   LIN {X 9.682, Y 0.522, Z 73.100}
   LaserStart_Ext()
   LIN {X -1.874, Y 0.522, Z 73.100}
   LaserEnd_Ext()
   LIN {X -2.025, Y -0.478, Z 73.100}
   LaserStart_Ext()
   LIN {X 9.715, Y -0.478, Z 73.100}
   LaserEnd_Ext()
   LIN {X 9.743, Y -1.478, Z 73.100}
   LaserStart_Ext()
   LIN {X -2.174, Y -1.478, Z 73.100}
   LaserEnd_Ext()
   LIN {X -2.322, Y -2.478, Z 73.100}
   LaserStart_Ext()
   LIN {X 9.770, Y -2.478, Z 73.100}
   LaserEnd_Ext()
   LIN {X 9.797, Y -3.478, Z 73.100}
   LaserStart_Ext()
   LIN {X -2.486, Y -3.478, Z 73.100}
   LaserEnd_Ext()
   LIN {X -2.718, Y -4.478, Z 73.100}
   LaserStart_Ext()
   LIN {X 9.824, Y -4.478, Z 73.100}
   LaserEnd_Ext()
   LIN {X 9.851, Y -5.478, Z 73.100}
   LaserStart_Ext()
   LIN {X -2.954, Y -5.478, Z 73.100}
   LaserEnd_Ext()
   LIN {X -3.189, Y -6.478, Z 73.100}
   LaserStart_Ext()
   LIN {X 9.859, Y -6.478, Z 73.100}
   LaserEnd_Ext()
   LIN {X 9.835, Y -7.478, Z 73.100}
   LaserStart_Ext()
   LIN {X -3.425, Y -7.478, Z 73.100}
   LaserEnd_Ext()
   LIN {X -3.704, Y -8.478, Z 73.100}
   LaserStart_Ext()
   LIN {X 9.811, Y -8.478, Z 73.100}
   LaserEnd_Ext()
   LIN {X 9.787, Y -9.478, Z 73.100}
   LaserStart_Ext()
   LIN {X -4.012, Y -9.478, Z 73.100}
   LaserEnd_Ext()
   LIN {X -4.320, Y -10.478, Z 73.100}
   LaserStart_Ext()
   LIN {X 9.763, Y -10.478, Z 73.100}
   LaserEnd_Ext()
   LIN {X 9.717, Y -11.478, Z 73.100}
   LaserStart_Ext()
   LIN {X -4.621, Y -11.478, Z 73.100}
   LaserEnd_Ext()
   LIN {X -4.914, Y -12.478, Z 73.100}
   LaserStart_Ext()
   LIN {X 9.656, Y -12.478, Z 73.100}
   LaserEnd_Ext()
   LIN {X 9.594, Y -13.478, Z 73.100}
   LaserStart_Ext()
   LIN {X -5.269, Y -13.478, Z 73.100}
   LaserEnd_Ext()
   LIN {X -5.652, Y -14.478, Z 73.100}
   LaserStart_Ext()
   LIN {X -1.831, Y -14.478, Z 73.100}
   LaserEnd_Ext()
   LIN {X 3.606, Y -14.478, Z 73.100}
   LaserStart_Ext()
   LIN {X 9.526, Y -14.478, Z 73.100}
   LaserEnd_Ext()
   LIN {X 9.435, Y -15.478, Z 73.100}
   LaserStart_Ext()
   LIN {X 5.099, Y -15.478, Z 73.100}
   LaserEnd_Ext()
   LIN {X -3.147, Y -15.478, Z 73.100}
   LaserStart_Ext()
   LIN {X -6.034, Y -15.478, Z 73.100}
   LaserEnd_Ext()
   LIN {X -6.409, Y -16.478, Z 73.100}
   LaserStart_Ext()
   LIN {X -4.119, Y -16.478, Z 73.100}
   LaserEnd_Ext()
   LIN {X 5.774, Y -16.478, Z 73.100}
   LaserStart_Ext()
   LIN {X 9.340, Y -16.478, Z 73.100}
   LaserEnd_Ext()
   LIN {X 9.248, Y -17.478, Z 73.100}
   LaserStart_Ext()
   LIN {X 6.448, Y -17.478, Z 73.100}
   LaserEnd_Ext()
   LIN {X -4.449, Y -17.478, Z 73.100}
   LaserStart_Ext()
   LIN {X -6.647, Y -17.478, Z 73.100}
   LaserEnd_Ext()
   LIN {X -6.866, Y -18.478, Z 73.100}
   LaserStart_Ext()
   LIN {X -4.737, Y -18.478, Z 73.100}
   LaserEnd_Ext()
   LIN {X 6.690, Y -18.478, Z 73.100}
   LaserStart_Ext()
   LIN {X 9.132, Y -18.478, Z 73.100}
   LaserEnd_Ext()
   LIN {X 9.008, Y -19.478, Z 73.100}
   LaserStart_Ext()
   LIN {X 6.800, Y -19.478, Z 73.100}
   LaserEnd_Ext()
   LIN {X -5.030, Y -19.478, Z 73.100}
   LaserStart_Ext()
   LIN {X -7.084, Y -19.478, Z 73.100}
   LaserEnd_Ext()
   LIN {X -6.914, Y -20.478, Z 73.100}
   LaserStart_Ext()
   LIN {X -4.983, Y -20.478, Z 73.100}
   LaserEnd_Ext()
   LIN {X 6.856, Y -20.478, Z 73.100}
   LaserStart_Ext()
   LIN {X 8.885, Y -20.478, Z 73.100}
   LaserEnd_Ext()
   LIN {X 8.615, Y -21.478, Z 73.100}
   LaserStart_Ext()
   LIN {X 6.497, Y -21.478, Z 73.100}
   LaserEnd_Ext()
   LIN {X -4.753, Y -21.478, Z 73.100}
   LaserStart_Ext()
   LIN {X -6.741, Y -21.478, Z 73.100}
   LaserEnd_Ext()
   LIN {X -6.568, Y -22.478, Z 73.100}
   LaserStart_Ext()
   LIN {X -4.439, Y -22.478, Z 73.100}
   LaserEnd_Ext()
   LIN {X 6.127, Y -22.478, Z 73.100}
   LaserStart_Ext()
   LIN {X 8.304, Y -22.478, Z 73.100}
   LaserEnd_Ext()
   LIN {X 7.905, Y -23.478, Z 73.100}
   LaserStart_Ext()
   LIN {X 5.494, Y -23.478, Z 73.100}
   LaserEnd_Ext()
   LIN {X -3.676, Y -23.478, Z 73.100}
   LaserStart_Ext()
   LIN {X -6.049, Y -23.478, Z 73.100}
   LaserEnd_Ext()
   LIN {X -5.411, Y -24.478, Z 73.100}
   LaserStart_Ext()
   LIN {X -2.745, Y -24.478, Z 73.100}
   LaserEnd_Ext()
   LIN {X 4.468, Y -24.478, Z 73.100}
   LaserStart_Ext()
   LIN {X 7.178, Y -24.478, Z 73.100}
   LaserEnd_Ext()
   LIN {X 6.380, Y -25.478, Z 73.100}
   LaserStart_Ext()
   LIN {X 2.288, Y -25.478, Z 73.100}
   LaserEnd_Ext()
   LIN {X -0.890, Y -25.478, Z 73.100}
   LaserStart_Ext()
   LIN {X -4.635, Y -25.478, Z 73.100}
   LaserEnd_Ext()
   LIN {X -3.321, Y -26.478, Z 73.100}
   LaserStart_Ext()
   LIN {X 4.795, Y -26.478, Z 73.100}
   LaserEnd_Ext()
   LIN {X 2.332, Y -27.478, Z 73.100}
   LaserStart_Ext()
   LIN {X -0.220, Y -27.478, Z 73.100}
   LaserEnd_Ext()
   LIN {X 5.714, Y -18.002, Z 73.950}
   LaserStart_Ext()
   LIN {X 5.782, Y -18.621, Z 73.950} C_DIS
   LIN {X 5.961, Y -20.198, Z 73.950} C_DIS
   LIN {X 5.569, Y -21.275, Z 73.950} C_DIS
   LIN {X 5.134, Y -22.450, Z 73.950} C_DIS
   LIN {X 3.676, Y -23.879, Z 73.950} C_DIS
   LIN {X 1.580, Y -24.646, Z 73.950} C_DIS
   LIN {X 0.264, Y -24.545, Z 73.950} C_DIS
   LIN {X -0.466, Y -24.486, Z 73.950} C_DIS
   LIN {X -1.367, Y -23.994, Z 73.950} C_DIS
   LIN {X -2.280, Y -23.497, Z 73.950} C_DIS
   LIN {X -2.814, Y -22.805, Z 73.950} C_DIS
   LIN {X -3.548, Y -21.845, Z 73.950} C_DIS
   LIN {X -3.815, Y -20.687, Z 73.950} C_DIS
   LIN {X -4.019, Y -19.812, Z 73.950} C_DIS
   LIN {X -3.359, Y -17.520, Z 73.950} C_DIS
   LIN {X -3.209, Y -16.978, Z 73.950} C_DIS
   LIN {X -2.651, Y -16.408, Z 73.950} C_DIS
   LIN {X -1.744, Y -15.500, Z 73.950} C_DIS
   LIN {X -0.780, Y -15.138, Z 73.950} C_DIS
   LIN {X 0.268, Y -14.732, Z 73.950} C_DIS
   LIN {X 1.745, Y -14.827, Z 73.950} C_DIS
   LIN {X 2.426, Y -14.872, Z 73.950} C_DIS
   LIN {X 2.906, Y -15.138, Z 73.950} C_DIS
   LIN {X 4.288, Y -15.897, Z 73.950} C_DIS
   LIN {X 5.367, Y -17.486, Z 73.950} C_DIS
   LIN {X 5.714, Y -18.002, Z 73.950}
   LaserEnd_Ext()
   LIN {X -4.465, Y 29.728, Z 73.950}
   LaserStart_Ext()
   LIN {X -4.338, Y 29.252, Z 73.950} C_DIS
   LIN {X -3.932, Y 27.798, Z 73.950} C_DIS
   LIN {X -3.385, Y 25.231, Z 73.950} C_DIS
   LIN {X -3.010, Y 22.795, Z 73.950} C_DIS
   LIN {X -2.537, Y 19.684, Z 73.950} C_DIS
   LIN {X -2.269, Y 17.163, Z 73.950} C_DIS
   LIN {X -2.334, Y 9.229, Z 73.950} C_DIS
   LIN {X -2.281, Y 5.034, Z 73.950} C_DIS
   LIN {X -2.382, Y 3.614, Z 73.950} C_DIS
   LIN {X -3.332, Y -2.684, Z 73.950} C_DIS
   LIN {X -3.464, Y -3.444, Z 73.950} C_DIS
   LIN {X -3.710, Y -4.444, Z 73.950} C_DIS
   LIN {X -4.539, Y -7.966, Z 73.950} C_DIS
   LIN {X -5.833, Y -12.173, Z 73.950} C_DIS
   LIN {X -5.930, Y -12.505, Z 73.950} C_DIS
   LIN {X -6.001, Y -12.710, Z 73.950} C_DIS
   LIN {X -6.189, Y -13.202, Z 73.950} C_DIS
   LIN {X -7.363, Y -16.331, Z 73.950} C_DIS
   LIN {X -7.756, Y -18.196, Z 73.950} C_DIS
   LIN {X -8.026, Y -19.431, Z 73.950} C_DIS
   LIN {X -7.590, Y -21.953, Z 73.950} C_DIS
   LIN {X -7.388, Y -23.087, Z 73.950} C_DIS
   LIN {X -7.016, Y -23.696, Z 73.950} C_DIS
   LIN {X -5.673, Y -25.799, Z 73.950} C_DIS
   LIN {X -4.232, Y -26.896, Z 73.950} C_DIS
   LIN {X -3.323, Y -27.631, Z 73.950} C_DIS
   LIN {X -2.826, Y -27.851, Z 73.950} C_DIS
   LIN {X 0.153, Y -28.583, Z 73.950} C_DIS
   LIN {X 0.920, Y -28.695, Z 73.950} C_DIS
   LIN {X 2.776, Y -28.357, Z 73.950} C_DIS
   LIN {X 4.021, Y -28.148, Z 73.950} C_DIS
   LIN {X 4.653, Y -27.762, Z 73.950} C_DIS
   LIN {X 7.309, Y -26.062, Z 73.950} C_DIS
   LIN {X 8.675, Y -24.178, Z 73.950} C_DIS
   LIN {X 9.048, Y -23.657, Z 73.950} C_DIS
   LIN {X 9.328, Y -22.743, Z 73.950} C_DIS
   LIN {X 9.923, Y -20.827, Z 73.950} C_DIS
   LIN {X 10.086, Y -19.502, Z 73.950} C_DIS
   LIN {X 10.310, Y -17.587, Z 73.950} C_DIS
   LIN {X 10.557, Y -14.882, Z 73.950} C_DIS
   LIN {X 10.580, Y -14.638, Z 73.950} C_DIS
   LIN {X 10.593, Y -14.454, Z 73.950} C_DIS
   LIN {X 10.811, Y -10.839, Z 73.950} C_DIS
   LIN {X 10.890, Y -7.567, Z 73.950} C_DIS
   LIN {X 10.916, Y -6.053, Z 73.950} C_DIS
   LIN {X 10.830, Y -3.422, Z 73.950} C_DIS
   LIN {X 10.724, Y 0.460, Z 73.950} C_DIS
   LIN {X 10.682, Y 1.154, Z 73.950} C_DIS
   LIN {X 10.578, Y 2.845, Z 73.950} C_DIS
   LIN {X 9.965, Y 8.271, Z 73.950} C_DIS
   LIN {X 9.810, Y 9.484, Z 73.950} C_DIS
   LIN {X 9.543, Y 10.719, Z 73.950} C_DIS
   LIN {X 7.636, Y 20.594, Z 73.950} C_DIS
   LIN {X 6.675, Y 24.247, Z 73.950} C_DIS
   LIN {X 5.389, Y 28.268, Z 73.950} C_DIS
   LIN {X 4.625, Y 30.707, Z 73.950} C_DIS
   LIN {X 3.858, Y 32.710, Z 73.950} C_DIS
   LIN {X 3.063, Y 34.855, Z 73.950} C_DIS
   LIN {X 2.554, Y 36.078, Z 73.950} C_DIS
   LIN {X 1.908, Y 37.651, Z 73.950} C_DIS
   LIN {X 0.727, Y 40.299, Z 73.950} C_DIS
   LIN {X 0.658, Y 40.450, Z 73.950} C_DIS
   LIN {X -0.114, Y 42.085, Z 73.950} C_DIS
   LIN {X -0.641, Y 43.162, Z 73.950} C_DIS
   LIN {X -0.767, Y 43.418, Z 73.950} C_DIS
   LIN {X -1.000, Y 43.725, Z 73.950} C_DIS
   LIN {X -1.653, Y 44.592, Z 73.950} C_DIS
   LIN {X -2.406, Y 45.027, Z 73.950} C_DIS
   LIN {X -3.161, Y 45.460, Z 73.950} C_DIS
   LIN {X -4.407, Y 45.564, Z 73.950} C_DIS
   LIN {X -4.900, Y 45.607, Z 73.950} C_DIS
   LIN {X -6.040, Y 44.979, Z 73.950} C_DIS
   LIN {X -7.379, Y 44.245, Z 73.950} C_DIS
   LIN {X -7.707, Y 43.622, Z 73.950} C_DIS
   LIN {X -8.206, Y 42.649, Z 73.950} C_DIS
   LIN {X -8.267, Y 41.850, Z 73.950} C_DIS
   LIN {X -8.311, Y 41.308, Z 73.950} C_DIS
   LIN {X -8.222, Y 40.974, Z 73.950} C_DIS
   LIN {X -7.991, Y 40.080, Z 73.950} C_DIS
   LIN {X -7.513, Y 38.929, Z 73.950} C_DIS
   LIN {X -6.918, Y 37.439, Z 73.950} C_DIS
   LIN {X -6.145, Y 35.340, Z 73.950} C_DIS
   LIN {X -6.099, Y 35.214, Z 73.950} C_DIS
   LIN {X -6.060, Y 35.097, Z 73.950} C_DIS
   LIN {X -5.193, Y 32.448, Z 73.950} C_DIS
   LIN {X -4.849, Y 31.163, Z 73.950} C_DIS
   LIN {X -4.593, Y 30.206, Z 73.950} C_DIS
   LIN {X -4.465, Y 29.728, Z 73.950}
   LaserEnd_Ext()
   LIN {X -7.280, Y 41.321, Z 73.950}
   LaserStart_Ext()
   LIN {X -7.280, Y 41.655, Z 73.950}
   LaserEnd_Ext()
   LIN {X -6.280, Y 43.707, Z 73.950}
   LaserStart_Ext()
   LIN {X -6.280, Y 38.538, Z 73.950}
   LaserEnd_Ext()
   LIN {X -6.280, Y -16.290, Z 73.950}
   LaserStart_Ext()
   LIN {X -6.280, Y -22.983, Z 73.950}
   LaserEnd_Ext()
   LIN {X -5.280, Y -24.557, Z 73.950}
   LaserStart_Ext()
   LIN {X -5.280, Y -13.624, Z 73.950}
   LaserEnd_Ext()
   LIN {X -5.280, Y 35.884, Z 73.950}
   LaserStart_Ext()
   LIN {X -5.280, Y 44.256, Z 73.950}
   LaserEnd_Ext()
   LIN {X -4.280, Y 44.550, Z 73.950}
   LaserStart_Ext()
   LIN {X -4.280, Y 32.874, Z 73.950}
   LaserEnd_Ext()
   LIN {X -4.280, Y -10.525, Z 73.950}
   LaserStart_Ext()
   LIN {X -4.280, Y -17.099, Z 73.950}
   LaserEnd_Ext()
   LIN {X -4.280, Y -22.535, Z 73.950}
   LaserStart_Ext()
   LIN {X -4.280, Y -25.603, Z 73.950}
   LaserEnd_Ext()
   LIN {X -3.280, Y -26.380, Z 73.950}
   LaserStart_Ext()
   LIN {X -3.280, Y -23.838, Z 73.950}
   LaserEnd_Ext()
   LIN {X -3.280, Y -15.623, Z 73.950}
   LaserStart_Ext()
   LIN {X -3.280, Y -6.982, Z 73.950}
   LaserEnd_Ext()
   LIN {X -3.280, Y 29.182, Z 73.950}
   LaserStart_Ext()
   LIN {X -3.280, Y 44.375, Z 73.950}
   LaserEnd_Ext()
   LIN {X -2.280, Y 43.762, Z 73.950}
   LaserStart_Ext()
   LIN {X -2.280, Y 24.625, Z 73.950}
   LaserEnd_Ext()
   LIN {X -2.280, Y -2.415, Z 73.950}
   LaserStart_Ext()
   LIN {X -2.280, Y -14.656, Z 73.950}
   LaserEnd_Ext()
   LIN {X -2.280, Y -24.636, Z 73.950}
   LaserStart_Ext()
   LIN {X -2.280, Y -26.955, Z 73.950}
   LaserEnd_Ext()
   LIN {X -1.280, Y -27.201, Z 73.950}
   LaserStart_Ext()
   LIN {X -1.280, Y -25.181, Z 73.950}
   LaserEnd_Ext()
   LIN {X -1.280, Y -14.257, Z 73.950}
   LaserStart_Ext()
   LIN {X -1.280, Y 15.884, Z 73.950}
   LaserEnd_Ext()
   LIN {X -1.280, Y 17.314, Z 73.950}
   LaserStart_Ext()
   LIN {X -1.280, Y 42.193, Z 73.950}
   LaserEnd_Ext()
   LIN {X -0.280, Y 40.094, Z 73.950}
   LaserStart_Ext()
   LIN {X -0.280, Y -13.872, Z 73.950}
   LaserEnd_Ext()
   LIN {X -0.280, Y -25.504, Z 73.950}
   LaserStart_Ext()
   LIN {X -0.280, Y -27.447, Z 73.950}
   LaserEnd_Ext()
   LIN {X 0.720, Y -27.655, Z 73.950}
   LaserStart_Ext()
   LIN {X 0.720, Y -25.583, Z 73.950}
   LaserEnd_Ext()
   LIN {X 0.720, Y -13.759, Z 73.950}
   LaserStart_Ext()
   LIN {X 0.720, Y 37.859, Z 73.950}
   LaserEnd_Ext()
   LIN {X 1.720, Y 35.480, Z 73.950}
   LaserStart_Ext()
   LIN {X 1.720, Y -13.823, Z 73.950}
   LaserEnd_Ext()
   LIN {X 1.720, Y -25.635, Z 73.950}
   LaserStart_Ext()
   LIN {X 1.720, Y -27.533, Z 73.950}
   LaserEnd_Ext()
   LIN {X 2.720, Y -27.352, Z 73.950}
   LaserStart_Ext()
   LIN {X 2.720, Y -25.298, Z 73.950}
   LaserEnd_Ext()
   LIN {X 2.720, Y -13.917, Z 73.950}
   LaserStart_Ext()
   LIN {X 2.720, Y 32.902, Z 73.950}
   LaserEnd_Ext()
   LIN {X 3.720, Y 30.251, Z 73.950}
   LaserStart_Ext()
   LIN {X 3.720, Y -14.444, Z 73.950}
   LaserEnd_Ext()
   LIN {X 3.720, Y -24.939, Z 73.950}
   LaserStart_Ext()
   LIN {X 3.720, Y -27.160, Z 73.950}
   LaserEnd_Ext()
   LIN {X 4.720, Y -26.532, Z 73.950}
   LaserStart_Ext()
   LIN {X 4.720, Y -24.256, Z 73.950}
   LaserEnd_Ext()
   LIN {X 4.720, Y -14.993, Z 73.950}
   LaserStart_Ext()
   LIN {X 4.720, Y 27.077, Z 73.950}
   LaserEnd_Ext()
   LIN {X 5.720, Y 23.946, Z 73.950}
   LaserStart_Ext()
   LIN {X 5.720, Y -16.226, Z 73.950}
   LaserEnd_Ext()
   LIN {X 5.720, Y -23.276, Z 73.950}
   LaserStart_Ext()
   LIN {X 5.720, Y -25.892, Z 73.950}
   LaserEnd_Ext()
   LIN {X 6.720, Y -25.171, Z 73.950}
   LaserStart_Ext()
   LIN {X 6.720, Y -21.036, Z 73.950}
   LaserEnd_Ext()
   LIN {X 6.720, Y -18.000, Z 73.950}
   LaserStart_Ext()
   LIN {X 6.720, Y 20.065, Z 73.950}
   LaserEnd_Ext()
   LIN {X 7.720, Y 14.884, Z 73.950}
   LaserStart_Ext()
   LIN {X 7.720, Y -23.791, Z 73.950}
   LaserEnd_Ext()
   LIN {X 8.720, Y -21.328, Z 73.950}
   LaserStart_Ext()
   LIN {X 8.720, Y 9.793, Z 73.950}
   LaserEnd_Ext()
   LIN {X 9.720, Y 0.498, Z 73.950}
   LaserStart_Ext()
   LIN {X 9.720, Y -12.314, Z 73.950}
   LaserEnd_Ext()
   LIN {X -3.144, Y -16.947, Z 74.800}
   LaserStart_Ext()
   LIN {X -1.831, Y -15.605, Z 74.800} C_DIS
   LIN {X -1.699, Y -15.468, Z 74.800} C_DIS
   LIN {X -1.436, Y -15.366, Z 74.800} C_DIS
   LIN {X 0.340, Y -14.679, Z 74.800} C_DIS
   LIN {X 1.732, Y -14.768, Z 74.800} C_DIS
   LIN {X 2.494, Y -14.814, Z 74.800} C_DIS
   LIN {X 3.293, Y -15.250, Z 74.800} C_DIS
   LIN {X 4.358, Y -15.835, Z 74.800} C_DIS
   LIN {X 5.158, Y -17.013, Z 74.800} C_DIS
   LIN {X 5.790, Y -17.936, Z 74.800} C_DIS
   LIN {X 5.889, Y -18.780, Z 74.800} C_DIS
   LIN {X 6.042, Y -20.132, Z 74.800} C_DIS
   LIN {X 5.244, Y -22.323, Z 74.800} C_DIS
   LIN {X 5.147, Y -22.457, Z 74.800} C_DIS
   LIN {X 3.744, Y -23.839, Z 74.800} C_DIS
   LIN {X 2.518, Y -24.284, Z 74.800} C_DIS
   LIN {X 1.668, Y -24.590, Z 74.800} C_DIS
   LIN {X 0.375, Y -24.491, Z 74.800} C_DIS
   LIN {X -0.375, Y -24.435, Z 74.800} C_DIS
   LIN {X -0.865, Y -24.171, Z 74.800} C_DIS
   LIN {X -2.192, Y -23.450, Z 74.800} C_DIS
   LIN {X -3.292, Y -22.022, Z 74.800} C_DIS
   LIN {X -3.464, Y -21.801, Z 74.800} C_DIS
   LIN {X -3.524, Y -21.549, Z 74.800} C_DIS
   LIN {X -3.940, Y -19.770, Z 74.800} C_DIS
   LIN {X -3.577, Y -18.513, Z 74.800} C_DIS
   LIN {X -3.144, Y -16.947, Z 74.800}
   LaserEnd_Ext()
   LIN {X -7.948, Y -19.398, Z 74.800}
   LaserStart_Ext()
   LIN {X -7.855, Y -19.936, Z 74.800} C_DIS
   LIN {X -7.301, Y -23.052, Z 74.800} C_DIS
   LIN {X -6.276, Y -24.727, Z 74.800} C_DIS
   LIN {X -5.697, Y -25.635, Z 74.800} C_DIS
   LIN {X -5.075, Y -26.108, Z 74.800} C_DIS
   LIN {X -3.295, Y -27.549, Z 74.800} C_DIS
   LIN {X -2.320, Y -27.979, Z 74.800} C_DIS
   LIN {X -0.748, Y -28.365, Z 74.800} C_DIS
   LIN {X 1.120, Y -28.639, Z 74.800} C_DIS
   LIN {X 3.648, Y -28.178, Z 74.800} C_DIS
   LIN {X 4.125, Y -28.085, Z 74.800} C_DIS
   LIN {X 5.363, Y -27.299, Z 74.800} C_DIS
   LIN {X 7.404, Y -25.993, Z 74.800} C_DIS
   LIN {X 8.053, Y -25.097, Z 74.800} C_DIS
   LIN {X 9.137, Y -23.583, Z 74.800} C_DIS
   LIN {X 9.950, Y -20.927, Z 74.800} C_DIS
   LIN {X 10.005, Y -20.752, Z 74.800} C_DIS
   LIN {X 10.020, Y -20.630, Z 74.800} C_DIS
   LIN {X 10.384, Y -17.510, Z 74.800} C_DIS
   LIN {X 10.556, Y -15.630, Z 74.800} C_DIS
   LIN {X 10.648, Y -14.561, Z 74.800} C_DIS
   LIN {X 10.747, Y -12.799, Z 74.800} C_DIS
   LIN {X 10.870, Y -10.762, Z 74.800} C_DIS
   LIN {X 10.909, Y -9.133, Z 74.800} C_DIS
   LIN {X 10.963, Y -5.975, Z 74.800} C_DIS
   LIN {X 10.784, Y -0.487, Z 74.800} C_DIS
   LIN {X 10.757, Y 0.537, Z 74.800} C_DIS
   LIN {X 10.745, Y 0.721, Z 74.800} C_DIS
   LIN {X 10.632, Y 2.561, Z 74.800} C_DIS
   LIN {X 10.112, Y 7.163, Z 74.800} C_DIS
   LIN {X 9.771, Y 9.841, Z 74.800} C_DIS
   LIN {X 9.180, Y 12.567, Z 74.800} C_DIS
   LIN {X 7.599, Y 20.760, Z 74.800} C_DIS
   LIN {X 6.801, Y 23.790, Z 74.800} C_DIS
   LIN {X 5.734, Y 27.126, Z 74.800} C_DIS
   LIN {X 4.623, Y 30.674, Z 74.800} C_DIS
   LIN {X 3.507, Y 33.588, Z 74.800} C_DIS
   LIN {X 3.024, Y 34.892, Z 74.800} C_DIS
   LIN {X 2.104, Y 37.104, Z 74.800} C_DIS
   LIN {X 1.928, Y 37.532, Z 74.800} C_DIS
   LIN {X 1.581, Y 38.309, Z 74.800} C_DIS
   LIN {X 0.644, Y 40.402, Z 74.800} C_DIS
   LIN {X -0.104, Y 41.979, Z 74.800} C_DIS
   LIN {X -0.179, Y 42.136, Z 74.800} C_DIS
   LIN {X -0.266, Y 42.313, Z 74.800} C_DIS
   LIN {X -0.835, Y 43.468, Z 74.800} C_DIS
   LIN {X -1.397, Y 44.210, Z 74.800} C_DIS
   LIN {X -1.724, Y 44.640, Z 74.800} C_DIS
   LIN {X -2.393, Y 45.022, Z 74.800} C_DIS
   LIN {X -3.234, Y 45.504, Z 74.800} C_DIS
   LIN {X -3.928, Y 45.563, Z 74.800} C_DIS
   LIN {X -4.973, Y 45.647, Z 74.800} C_DIS
   LIN {X -6.690, Y 44.715, Z 74.800} C_DIS
   LIN {X -7.418, Y 44.316, Z 74.800} C_DIS
   LIN {X -7.716, Y 43.749, Z 74.800} C_DIS
   LIN {X -8.254, Y 42.753, Z 74.800} C_DIS
   LIN {X -8.323, Y 41.939, Z 74.800} C_DIS
   LIN {X -8.372, Y 41.322, Z 74.800} C_DIS
   LIN {X -8.169, Y 40.552, Z 74.800} C_DIS
   LIN {X -8.051, Y 40.112, Z 74.800} C_DIS
   LIN {X -7.913, Y 39.782, Z 74.800} C_DIS
   LIN {X -7.568, Y 38.959, Z 74.800} C_DIS
   LIN {X -7.062, Y 37.699, Z 74.800} C_DIS
   LIN {X -6.972, Y 37.474, Z 74.800} C_DIS
   LIN {X -6.886, Y 37.245, Z 74.800} C_DIS
   LIN {X -6.148, Y 35.252, Z 74.800} C_DIS
   LIN {X -5.378, Y 32.924, Z 74.800} C_DIS
   LIN {X -5.235, Y 32.487, Z 74.800} C_DIS
   LIN {X -5.179, Y 32.276, Z 74.800} C_DIS
   LIN {X -4.827, Y 30.959, Z 74.800} C_DIS
   LIN {X -4.651, Y 30.303, Z 74.800} C_DIS
   LIN {X -4.475, Y 29.647, Z 74.800} C_DIS
   LIN {X -3.917, Y 27.648, Z 74.800} C_DIS
   LIN {X -3.438, Y 25.397, Z 74.800} C_DIS
   LIN {X -2.758, Y 20.982, Z 74.800} C_DIS
   LIN {X -2.456, Y 18.992, Z 74.800} C_DIS
   LIN {X -2.284, Y 17.379, Z 74.800} C_DIS
   LIN {X -2.326, Y 12.303, Z 74.800} C_DIS
   LIN {X -2.239, Y 5.526, Z 74.800} C_DIS
   LIN {X -2.403, Y 3.231, Z 74.800} C_DIS
   LIN {X -3.187, Y -1.972, Z 74.800} C_DIS
   LIN {X -3.508, Y -3.811, Z 74.800} C_DIS
   LIN {X -4.102, Y -6.230, Z 74.800} C_DIS
   LIN {X -4.597, Y -8.330, Z 74.800} C_DIS
   LIN {X -5.563, Y -11.471, Z 74.800} C_DIS
   LIN {X -5.912, Y -12.599, Z 74.800} C_DIS
   LIN {X -6.221, Y -13.443, Z 74.800} C_DIS
   LIN {X -7.292, Y -16.296, Z 74.800} C_DIS
   LIN {X -7.890, Y -19.135, Z 74.800} C_DIS
   LIN {X -7.948, Y -19.398, Z 74.800}
   LaserEnd_Ext()
   LIN {X -0.648, Y -27.360, Z 74.800}
   LaserStart_Ext()
   LIN {X 2.557, Y -27.360, Z 74.800}
   LaserEnd_Ext()
   LIN {X 4.975, Y -26.360, Z 74.800}
   LaserStart_Ext()
   LIN {X -3.174, Y -26.360, Z 74.800}
   LaserEnd_Ext()
   LIN {X -4.410, Y -25.360, Z 74.800}
   LaserStart_Ext()
   LIN {X -0.756, Y -25.360, Z 74.800}
   LaserEnd_Ext()
   LIN {X 2.482, Y -25.360, Z 74.800}
   LaserStart_Ext()
   LIN {X 6.537, Y -25.360, Z 74.800}
   LaserEnd_Ext()
   LIN {X 7.351, Y -24.360, Z 74.800}
   LaserStart_Ext()
   LIN {X 4.640, Y -24.360, Z 74.800}
   LaserEnd_Ext()
   LIN {X -2.612, Y -24.360, Z 74.800}
   LaserStart_Ext()
   LIN {X -5.325, Y -24.360, Z 74.800}
   LaserEnd_Ext()
   LIN {X -5.940, Y -23.360, Z 74.800}
   LaserStart_Ext()
   LIN {X -3.524, Y -23.360, Z 74.800}
   LaserEnd_Ext()
   LIN {X 5.655, Y -23.360, Z 74.800}
   LaserStart_Ext()
   LIN {X 8.067, Y -23.360, Z 74.800}
   LaserEnd_Ext()
   LIN {X 8.466, Y -22.360, Z 74.800}
   LaserStart_Ext()
   LIN {X 6.295, Y -22.360, Z 74.800}
   LaserEnd_Ext()
   LIN {X -4.292, Y -22.360, Z 74.800}
   LaserStart_Ext()
   LIN {X -6.408, Y -22.360, Z 74.800}
   LaserEnd_Ext()
   LIN {X -6.586, Y -21.360, Z 74.800}
   LaserStart_Ext()
   LIN {X -4.595, Y -21.360, Z 74.800}
   LaserEnd_Ext()
   LIN {X 6.659, Y -21.360, Z 74.800}
   LaserStart_Ext()
   LIN {X 8.772, Y -21.360, Z 74.800}
   LaserEnd_Ext()
   LIN {X 9.045, Y -20.360, Z 74.800}
   LaserStart_Ext()
   LIN {X 7.014, Y -20.360, Z 74.800}
   LaserEnd_Ext()
   LIN {X -4.829, Y -20.360, Z 74.800}
   LaserStart_Ext()
   LIN {X -6.764, Y -20.360, Z 74.800}
   LaserEnd_Ext()
   LIN {X -6.916, Y -19.360, Z 74.800}
   LaserStart_Ext()
   LIN {X -4.862, Y -19.360, Z 74.800}
   LaserEnd_Ext()
   LIN {X 6.961, Y -19.360, Z 74.800}
   LaserStart_Ext()
   LIN {X 9.161, Y -19.360, Z 74.800}
   LaserEnd_Ext()
   LIN {X 9.278, Y -18.360, Z 74.800}
   LaserStart_Ext()
   LIN {X 6.846, Y -18.360, Z 74.800}
   LaserEnd_Ext()
   LIN {X -4.574, Y -18.360, Z 74.800}
   LaserStart_Ext()
   LIN {X -6.705, Y -18.360, Z 74.800}
   LaserEnd_Ext()
   LIN {X -6.494, Y -17.360, Z 74.800}
   LaserStart_Ext()
   LIN {X -4.296, Y -17.360, Z 74.800}
   LaserEnd_Ext()
   LIN {X 6.608, Y -17.360, Z 74.800}
   LaserStart_Ext()
   LIN {X 9.394, Y -17.360, Z 74.800}
   LaserEnd_Ext()
   LIN {X 9.485, Y -16.360, Z 74.800}
   LaserStart_Ext()
   LIN {X 5.924, Y -16.360, Z 74.800}
   LaserEnd_Ext()
   LIN {X -3.952, Y -16.360, Z 74.800}
   LaserStart_Ext()
   LIN {X -6.248, Y -16.360, Z 74.800}
   LaserEnd_Ext()
   LIN {X -5.873, Y -15.360, Z 74.800}
   LaserStart_Ext()
   LIN {X -2.991, Y -15.360, Z 74.800}
   LaserEnd_Ext()
   LIN {X 5.245, Y -15.360, Z 74.800}
   LaserStart_Ext()
   LIN {X 9.576, Y -15.360, Z 74.800}
   LaserEnd_Ext()
   LIN {X 9.658, Y -14.360, Z 74.800}
   LaserStart_Ext()
   LIN {X 3.750, Y -14.360, Z 74.800}
   LaserEnd_Ext()
   LIN {X -1.608, Y -14.360, Z 74.800}
   LaserStart_Ext()
   LIN {X -5.498, Y -14.360, Z 74.800}
   LaserEnd_Ext()
   LIN {X -5.126, Y -13.360, Z 74.800}
   LaserStart_Ext()
   LIN {X 9.714, Y -13.360, Z 74.800}
   LaserEnd_Ext()
   LIN {X 9.771, Y -12.360, Z 74.800}
   LaserStart_Ext()
   LIN {X -4.791, Y -12.360, Z 74.800}
   LaserEnd_Ext()
   LIN {X -4.482, Y -11.360, Z 74.800}
   LaserStart_Ext()
   LIN {X 9.832, Y -11.360, Z 74.800}
   LaserEnd_Ext()
   LIN {X 9.879, Y -10.360, Z 74.800}
   LaserStart_Ext()
   LIN {X -4.175, Y -10.360, Z 74.800}
   LaserEnd_Ext()
   LIN {X -3.867, Y -9.360, Z 74.800}
   LaserStart_Ext()
   LIN {X 9.903, Y -9.360, Z 74.800}
   LaserEnd_Ext()
   LIN {X 9.922, Y -8.360, Z 74.800}
   LaserStart_Ext()
   LIN {X -3.576, Y -8.360, Z 74.800}
   LaserEnd_Ext()
   LIN {X -3.341, Y -7.360, Z 74.800}
   LaserStart_Ext()
   LIN {X 9.939, Y -7.360, Z 74.800}
   LaserEnd_Ext()
   LIN {X 9.956, Y -6.360, Z 74.800}
   LaserStart_Ext()
   LIN {X -3.105, Y -6.360, Z 74.800}
   LaserEnd_Ext()
   LIN {X -2.859, Y -5.360, Z 74.800}
   LaserStart_Ext()
   LIN {X 9.942, Y -5.360, Z 74.800}
   LaserEnd_Ext()
   LIN {X 9.910, Y -4.360, Z 74.800}
   LaserStart_Ext()
   LIN {X -2.613, Y -4.360, Z 74.800}
   LaserEnd_Ext()
   LIN {X -2.414, Y -3.360, Z 74.800}
   LaserStart_Ext()
   LIN {X 9.877, Y -3.360, Z 74.800}
   LaserEnd_Ext()
   LIN {X 9.845, Y -2.360, Z 74.800}
   LaserStart_Ext()
   LIN {X -2.240, Y -2.360, Z 74.800}
   LaserEnd_Ext()
   LIN {X -2.084, Y -1.360, Z 74.800}
   LaserStart_Ext()
   LIN {X 9.812, Y -1.360, Z 74.800}
   LaserEnd_Ext()
   LIN {X 9.781, Y -0.360, Z 74.800}
   LaserStart_Ext()
   LIN {X -1.933, Y -0.360, Z 74.800}
   LaserEnd_Ext()
   LIN {X -1.782, Y 0.640, Z 74.800}
   LaserStart_Ext()
   LIN {X 9.748, Y 0.640, Z 74.800}
   LaserEnd_Ext()
   LIN {X 9.687, Y 1.640, Z 74.800}
   LaserStart_Ext()
   LIN {X -1.632, Y 1.640, Z 74.800}
   LaserEnd_Ext()
   LIN {X -1.481, Y 2.640, Z 74.800}
   LaserStart_Ext()
   LIN {X 9.617, Y 2.640, Z 74.800}
   LaserEnd_Ext()
   LIN {X 9.504, Y 3.640, Z 74.800}
   LaserStart_Ext()
   LIN {X -1.371, Y 3.640, Z 74.800}
   LaserEnd_Ext()
   LIN {X -1.300, Y 4.640, Z 74.800}
   LaserStart_Ext()
   LIN {X 9.391, Y 4.640, Z 74.800}
   LaserEnd_Ext()
   LIN {X 9.278, Y 5.640, Z 74.800}
   LaserStart_Ext()
   LIN {X -1.241, Y 5.640, Z 74.800}
   LaserEnd_Ext()
   LIN {X -1.254, Y 6.640, Z 74.800}
   LaserStart_Ext()
   LIN {X 9.165, Y 6.640, Z 74.800}
   LaserEnd_Ext()
   LIN {X 9.044, Y 7.640, Z 74.800}
   LaserStart_Ext()
   LIN {X -1.266, Y 7.640, Z 74.800}
   LaserEnd_Ext()
   LIN {X -1.279, Y 8.640, Z 74.800}
   LaserStart_Ext()
   LIN {X 8.916, Y 8.640, Z 74.800}
   LaserEnd_Ext()
   LIN {X 8.789, Y 9.640, Z 74.800}
   LaserStart_Ext()
   LIN {X -1.292, Y 9.640, Z 74.800}
   LaserEnd_Ext()
   LIN {X -1.305, Y 10.640, Z 74.800}
   LaserStart_Ext()
   LIN {X 8.575, Y 10.640, Z 74.800}
   LaserEnd_Ext()
   LIN {X 8.358, Y 11.640, Z 74.800}
   LaserStart_Ext()
   LIN {X -1.317, Y 11.640, Z 74.800}
   LaserEnd_Ext()
   LIN {X -1.323, Y 12.640, Z 74.800}
   LaserStart_Ext()
   LIN {X 8.147, Y 12.640, Z 74.800}
   LaserEnd_Ext()
   LIN {X 7.954, Y 13.640, Z 74.800}
   LaserStart_Ext()
   LIN {X -1.315, Y 13.640, Z 74.800}
   LaserEnd_Ext()
   LIN {X -1.307, Y 14.640, Z 74.800}
   LaserStart_Ext()
   LIN {X 7.761, Y 14.640, Z 74.800}
   LaserEnd_Ext()
   LIN {X 7.568, Y 15.640, Z 74.800}
   LaserStart_Ext()
   LIN {X -1.298, Y 15.640, Z 74.800}
   LaserEnd_Ext()
   LIN {X -1.290, Y 16.640, Z 74.800}
   LaserStart_Ext()
   LIN {X 7.375, Y 16.640, Z 74.800}
   LaserEnd_Ext()
   LIN {X 7.182, Y 17.640, Z 74.800}
   LaserStart_Ext()
   LIN {X -1.306, Y 17.640, Z 74.800}
   LaserEnd_Ext()
   LIN {X -1.413, Y 18.640, Z 74.800}
   LaserStart_Ext()
   LIN {X 6.989, Y 18.640, Z 74.800}
   LaserEnd_Ext()
   LIN {X 6.796, Y 19.640, Z 74.800}
   LaserStart_Ext()
   LIN {X -1.543, Y 19.640, Z 74.800}
   LaserEnd_Ext()
   LIN {X -1.695, Y 20.640, Z 74.800}
   LaserStart_Ext()
   LIN {X 6.596, Y 20.640, Z 74.800}
   LaserEnd_Ext()
   LIN {X 6.333, Y 21.640, Z 74.800}
   LaserStart_Ext()
   LIN {X -1.847, Y 21.640, Z 74.800}
   LaserEnd_Ext()
   LIN {X -2.001, Y 22.640, Z 74.800}
   LaserStart_Ext()
   LIN {X 6.070, Y 22.640, Z 74.800}
   LaserEnd_Ext()
   LIN {X 5.799, Y 23.640, Z 74.800}
   LaserStart_Ext()
   LIN {X -2.155, Y 23.640, Z 74.800}
   LaserEnd_Ext()
   LIN {X -2.309, Y 24.640, Z 74.800}
   LaserStart_Ext()
   LIN {X 5.479, Y 24.640, Z 74.800}
   LaserEnd_Ext()
   LIN {X 5.160, Y 25.640, Z 74.800}
   LaserStart_Ext()
   LIN {X -2.467, Y 25.640, Z 74.800}
   LaserEnd_Ext()
   LIN {X -2.680, Y 26.640, Z 74.800}
   LaserStart_Ext()
   LIN {X 4.840, Y 26.640, Z 74.800}
   LaserEnd_Ext()
   LIN {X 4.525, Y 27.640, Z 74.800}
   LaserStart_Ext()
   LIN {X -2.893, Y 27.640, Z 74.800}
   LaserEnd_Ext()
   LIN {X -3.156, Y 28.640, Z 74.800}
   LaserStart_Ext()
   LIN {X 4.212, Y 28.640, Z 74.800}
   LaserEnd_Ext()
   LIN {X 3.899, Y 29.640, Z 74.800}
   LaserStart_Ext()
   LIN {X -3.435, Y 29.640, Z 74.800}
   LaserEnd_Ext()
   LIN {X -3.706, Y 30.640, Z 74.800}
   LaserStart_Ext()
   LIN {X 3.565, Y 30.640, Z 74.800}
   LaserEnd_Ext()
   LIN {X 3.182, Y 31.640, Z 74.800}
   LaserStart_Ext()
   LIN {X -3.973, Y 31.640, Z 74.800}
   LaserEnd_Ext()
   LIN {X -4.241, Y 32.640, Z 74.800}
   LaserStart_Ext()
   LIN {X 2.799, Y 32.640, Z 74.800}
   LaserEnd_Ext()
   LIN {X 2.421, Y 33.640, Z 74.800}
   LaserStart_Ext()
   LIN {X -4.562, Y 33.640, Z 74.800}
   LaserEnd_Ext()
   LIN {X -4.892, Y 34.640, Z 74.800}
   LaserStart_Ext()
   LIN {X 2.045, Y 34.640, Z 74.800}
   LaserEnd_Ext()
   LIN {X 1.629, Y 35.640, Z 74.800}
   LaserStart_Ext()
   LIN {X -5.225, Y 35.640, Z 74.800}
   LaserEnd_Ext()
   LIN {X -5.596, Y 36.640, Z 74.800}
   LaserStart_Ext()
   LIN {X 1.214, Y 36.640, Z 74.800}
   LaserEnd_Ext()
   LIN {X 0.785, Y 37.640, Z 74.800}
   LaserStart_Ext()
   LIN {X -5.966, Y 37.640, Z 74.800}
   LaserEnd_Ext()
   LIN {X -6.363, Y 38.640, Z 74.800}
   LaserStart_Ext()
   LIN {X 0.337, Y 38.640, Z 74.800}
   LaserEnd_Ext()
   LIN {X -0.110, Y 39.640, Z 74.800}
   LaserStart_Ext()
   LIN {X -6.769, Y 39.640, Z 74.800}
   LaserEnd_Ext()
   LIN {X -7.157, Y 40.640, Z 74.800}
   LaserStart_Ext()
   LIN {X -0.576, Y 40.640, Z 74.800}
   LaserEnd_Ext()
   LIN {X -1.050, Y 41.640, Z 74.800}
   LaserStart_Ext()
   LIN {X -7.344, Y 41.640, Z 74.800}
   LaserEnd_Ext()
   LIN {X -7.178, Y 42.640, Z 74.800}
   LaserStart_Ext()
   LIN {X -1.542, Y 42.640, Z 74.800}
   LaserEnd_Ext()
   LIN {X -2.220, Y 43.640, Z 74.800}
   LaserStart_Ext()
   LIN {X -6.571, Y 43.640, Z 74.800}
   LaserEnd_Ext()
   LIN {X -2.103, Y -23.404, Z 75.650}
   LaserStart_Ext()
   LIN {X -2.213, Y -23.262, Z 75.650} C_DIS
   LIN {X -3.379, Y -21.757, Z 75.650} C_DIS
   LIN {X -3.787, Y -20.040, Z 75.650} C_DIS
   LIN {X -3.860, Y -19.727, Z 75.650} C_DIS
   LIN {X -3.796, Y -19.506, Z 75.650} C_DIS
   LIN {X -3.080, Y -16.916, Z 75.650} C_DIS
   LIN {X -2.588, Y -16.414, Z 75.650} C_DIS
   LIN {X -1.625, Y -15.418, Z 75.650} C_DIS
   LIN {X 0.285, Y -14.675, Z 75.650} C_DIS
   LIN {X 0.412, Y -14.626, Z 75.650} C_DIS
   LIN {X 2.562, Y -14.757, Z 75.650} C_DIS
   LIN {X 4.181, Y -15.638, Z 75.650} C_DIS
   LIN {X 4.429, Y -15.772, Z 75.650} C_DIS
   LIN {X 4.624, Y -16.056, Z 75.650} C_DIS
   LIN {X 5.866, Y -17.870, Z 75.650} C_DIS
   LIN {X 6.121, Y -20.057, Z 75.650} C_DIS
   LIN {X 5.310, Y -22.316, Z 75.650} C_DIS
   LIN {X 4.490, Y -23.131, Z 75.650} C_DIS
   LIN {X 3.832, Y -23.779, Z 75.650} C_DIS
   LIN {X 2.338, Y -24.322, Z 75.650} C_DIS
   LIN {X 1.757, Y -24.535, Z 75.650} C_DIS
   LIN {X 1.378, Y -24.508, Z 75.650} C_DIS
   LIN {X -0.284, Y -24.384, Z 75.650} C_DIS
   LIN {X -1.971, Y -23.476, Z 75.650} C_DIS
   LIN {X -2.103, Y -23.404, Z 75.650}
   LaserEnd_Ext()
   LIN {X -8.316, Y 42.672, Z 75.650}
   LaserStart_Ext()
   LIN {X -8.439, Y 41.409, Z 75.650} C_DIS
   LIN {X -8.249, Y 40.656, Z 75.650} C_DIS
   LIN {X -8.112, Y 40.145, Z 75.650} C_DIS
   LIN {X -7.849, Y 39.519, Z 75.650} C_DIS
   LIN {X -7.626, Y 38.993, Z 75.650} C_DIS
   LIN {X -7.470, Y 38.609, Z 75.650} C_DIS
   LIN {X -7.026, Y 37.510, Z 75.650} C_DIS
   LIN {X -6.217, Y 35.345, Z 75.650} C_DIS
   LIN {X -6.165, Y 35.193, Z 75.650} C_DIS
   LIN {X -5.278, Y 32.527, Z 75.650} C_DIS
   LIN {X -5.060, Y 31.713, Z 75.650} C_DIS
   LIN {X -4.613, Y 30.043, Z 75.650} C_DIS
   LIN {X -3.902, Y 27.497, Z 75.650} C_DIS
   LIN {X -3.490, Y 25.563, Z 75.650} C_DIS
   LIN {X -2.506, Y 19.169, Z 75.650} C_DIS
   LIN {X -2.374, Y 18.299, Z 75.650} C_DIS
   LIN {X -2.299, Y 17.595, Z 75.650} C_DIS
   LIN {X -2.317, Y 15.378, Z 75.650} C_DIS
   LIN {X -2.198, Y 6.017, Z 75.650} C_DIS
   LIN {X -2.424, Y 2.848, Z 75.650} C_DIS
   LIN {X -3.043, Y -1.261, Z 75.650} C_DIS
   LIN {X -3.551, Y -4.178, Z 75.650} C_DIS
   LIN {X -4.495, Y -8.017, Z 75.650} C_DIS
   LIN {X -4.654, Y -8.694, Z 75.650} C_DIS
   LIN {X -4.966, Y -9.707, Z 75.650} C_DIS
   LIN {X -5.846, Y -12.554, Z 75.650} C_DIS
   LIN {X -6.628, Y -14.681, Z 75.650} C_DIS
   LIN {X -7.220, Y -16.261, Z 75.650} C_DIS
   LIN {X -7.632, Y -18.216, Z 75.650} C_DIS
   LIN {X -7.869, Y -19.365, Z 75.650} C_DIS
   LIN {X -7.699, Y -20.288, Z 75.650} C_DIS
   LIN {X -7.214, Y -23.017, Z 75.650} C_DIS
   LIN {X -5.847, Y -25.252, Z 75.650} C_DIS
   LIN {X -5.693, Y -25.501, Z 75.650} C_DIS
   LIN {X -5.431, Y -25.715, Z 75.650} C_DIS
   LIN {X -3.266, Y -27.466, Z 75.650} C_DIS
   LIN {X -1.815, Y -28.107, Z 75.650} C_DIS
   LIN {X -1.648, Y -28.148, Z 75.650} C_DIS
   LIN {X 1.320, Y -28.582, Z 75.650} C_DIS
   LIN {X 2.776, Y -28.317, Z 75.650} C_DIS
   LIN {X 4.147, Y -28.051, Z 75.650} C_DIS
   LIN {X 7.391, Y -25.991, Z 75.650} C_DIS
   LIN {X 7.493, Y -25.929, Z 75.650} C_DIS
   LIN {X 7.598, Y -25.782, Z 75.650} C_DIS
   LIN {X 9.226, Y -23.509, Z 75.650} C_DIS
   LIN {X 9.768, Y -21.738, Z 75.650} C_DIS
   LIN {X 10.087, Y -20.676, Z 75.650} C_DIS
   LIN {X 10.323, Y -18.602, Z 75.650} C_DIS
   LIN {X 10.459, Y -17.433, Z 75.650} C_DIS
   LIN {X 10.517, Y -16.801, Z 75.650} C_DIS
   LIN {X 10.715, Y -14.483, Z 75.650} C_DIS
   LIN {X 10.928, Y -10.696, Z 75.650} C_DIS
   LIN {X 11.010, Y -5.897, Z 75.650} C_DIS
   LIN {X 10.842, Y -0.735, Z 75.650} C_DIS
   LIN {X 10.789, Y 0.615, Z 75.650} C_DIS
   LIN {X 10.687, Y 2.276, Z 75.650} C_DIS
   LIN {X 10.260, Y 6.056, Z 75.650} C_DIS
   LIN {X 9.732, Y 10.198, Z 75.650} C_DIS
   LIN {X 8.817, Y 14.415, Z 75.650} C_DIS
   LIN {X 7.561, Y 20.926, Z 75.650} C_DIS
   LIN {X 6.927, Y 23.334, Z 75.650} C_DIS
   LIN {X 6.079, Y 25.985, Z 75.650} C_DIS
   LIN {X 4.620, Y 30.642, Z 75.650} C_DIS
   LIN {X 3.155, Y 34.466, Z 75.650} C_DIS
   LIN {X 2.984, Y 34.929, Z 75.650} C_DIS
   LIN {X 2.482, Y 36.135, Z 75.650} C_DIS
   LIN {X 1.907, Y 37.509, Z 75.650} C_DIS
   LIN {X 0.693, Y 40.211, Z 75.650} C_DIS
   LIN {X 0.585, Y 40.451, Z 75.650} C_DIS
   LIN {X -0.242, Y 42.184, Z 75.650} C_DIS
   LIN {X -0.732, Y 43.173, Z 75.650} C_DIS
   LIN {X -0.904, Y 43.517, Z 75.650} C_DIS
   LIN {X -1.175, Y 43.872, Z 75.650} C_DIS
   LIN {X -1.795, Y 44.687, Z 75.650} C_DIS
   LIN {X -2.682, Y 45.194, Z 75.650} C_DIS
   LIN {X -3.307, Y 45.549, Z 75.650} C_DIS
   LIN {X -4.824, Y 45.669, Z 75.650} C_DIS
   LIN {X -5.046, Y 45.687, Z 75.650} C_DIS
   LIN {X -5.280, Y 45.560, Z 75.650} C_DIS
   LIN {X -7.456, Y 44.387, Z 75.650} C_DIS
   LIN {X -8.215, Y 43.016, Z 75.650} C_DIS
   LIN {X -8.300, Y 42.857, Z 75.650} C_DIS
   LIN {X -8.316, Y 42.672, Z 75.650}
   LaserEnd_Ext()
   LIN {X 9.602, Y -15.765, Z 75.650}
   LaserStart_Ext()
   LIN {X 9.602, Y 2.970, Z 75.650}
   LaserEnd_Ext()
   LIN {X 8.602, Y 10.690, Z 75.650}
   LaserStart_Ext()
   LIN {X 8.602, Y -22.132, Z 75.650}
   LaserEnd_Ext()
   LIN {X 7.602, Y -24.060, Z 75.650}
   LaserStart_Ext()
   LIN {X 7.602, Y 15.436, Z 75.650}
   LaserEnd_Ext()
   LIN {X 6.602, Y 20.617, Z 75.650}
   LaserStart_Ext()
   LIN {X 6.602, Y -17.176, Z 75.650}
   LaserEnd_Ext()
   LIN {X 6.602, Y -21.682, Z 75.650}
   LaserStart_Ext()
   LIN {X 6.602, Y -25.307, Z 75.650}
   LaserEnd_Ext()
   LIN {X 5.602, Y -25.942, Z 75.650}
   LaserStart_Ext()
   LIN {X 5.602, Y -23.436, Z 75.650}
   LaserEnd_Ext()
   LIN {X 5.602, Y -15.714, Z 75.650}
   LaserStart_Ext()
   LIN {X 5.602, Y 24.194, Z 75.650}
   LaserEnd_Ext()
   LIN {X 4.602, Y 27.355, Z 75.650}
   LaserStart_Ext()
   LIN {X 4.602, Y -14.729, Z 75.650}
   LaserEnd_Ext()
   LIN {X 4.602, Y -24.424, Z 75.650}
   LaserStart_Ext()
   LIN {X 4.602, Y -26.578, Z 75.650}
   LaserEnd_Ext()
   LIN {X 3.602, Y -27.138, Z 75.650}
   LaserStart_Ext()
   LIN {X 3.602, Y -24.927, Z 75.650}
   LaserEnd_Ext()
   LIN {X 3.602, Y -14.184, Z 75.650}
   LaserStart_Ext()
   LIN {X 3.602, Y 30.505, Z 75.650}
   LaserEnd_Ext()
   LIN {X 2.602, Y 33.116, Z 75.650}
   LaserStart_Ext()
   LIN {X 2.602, Y -13.757, Z 75.650}
   LaserEnd_Ext()
   LIN {X 2.602, Y -25.290, Z 75.650}
   LaserStart_Ext()
   LIN {X 2.602, Y -27.332, Z 75.650}
   LaserEnd_Ext()
   LIN {X 1.602, Y -27.514, Z 75.650}
   LaserStart_Ext()
   LIN {X 1.602, Y -25.526, Z 75.650}
   LaserEnd_Ext()
   LIN {X 1.602, Y -13.696, Z 75.650}
   LaserStart_Ext()
   LIN {X 1.602, Y 35.648, Z 75.650}
   LaserEnd_Ext()
   LIN {X 0.602, Y 37.974, Z 75.650}
   LaserStart_Ext()
   LIN {X 0.602, Y -13.636, Z 75.650}
   LaserEnd_Ext()
   LIN {X 0.602, Y -25.453, Z 75.650}
   LaserStart_Ext()
   LIN {X 0.602, Y -27.466, Z 75.650}
   LaserEnd_Ext()
   LIN {X -0.398, Y -27.320, Z 75.650}
   LaserStart_Ext()
   LIN {X -0.398, Y -25.376, Z 75.650}
   LaserEnd_Ext()
   LIN {X -0.398, Y -13.868, Z 75.650}
   LaserStart_Ext()
   LIN {X -0.398, Y 40.190, Z 75.650}
   LaserEnd_Ext()
   LIN {X -1.398, Y 42.265, Z 75.650}
   LaserStart_Ext()
   LIN {X -1.398, Y 18.534, Z 75.650}
   LaserEnd_Ext()
   LIN {X -1.398, Y 3.175, Z 75.650}
   LaserStart_Ext()
   LIN {X -1.398, Y -14.256, Z 75.650}
   LaserEnd_Ext()
   LIN {X -1.398, Y -24.920, Z 75.650}
   LaserStart_Ext()
   LIN {X -1.398, Y -27.174, Z 75.650}
   LaserEnd_Ext()
   LIN {X -2.398, Y -26.757, Z 75.650}
   LaserStart_Ext()
   LIN {X -2.398, Y -24.381, Z 75.650}
   LaserEnd_Ext()
   LIN {X -2.398, Y -14.778, Z 75.650}
   LaserStart_Ext()
   LIN {X -2.398, Y -3.384, Z 75.650}
   LaserEnd_Ext()
   LIN {X -2.398, Y 25.041, Z 75.650}
   LaserStart_Ext()
   LIN {X -2.398, Y 43.828, Z 75.650}
   LaserEnd_Ext()
   LIN {X -3.398, Y 44.451, Z 75.650}
   LaserStart_Ext()
   LIN {X -3.398, Y 29.410, Z 75.650}
   LaserEnd_Ext()
   LIN {X -3.398, Y -7.743, Z 75.650}
   LaserStart_Ext()
   LIN {X -3.398, Y -15.811, Z 75.650}
   LaserEnd_Ext()
   LIN {X -3.398, Y -23.365, Z 75.650}
   LaserStart_Ext()
   LIN {X -3.398, Y -26.073, Z 75.650}
   LaserEnd_Ext()
   LIN {X -4.398, Y -25.264, Z 75.650}
   LaserStart_Ext()
   LIN {X -4.398, Y -21.795, Z 75.650}
   LaserEnd_Ext()
   LIN {X -4.398, Y -17.931, Z 75.650}
   LaserStart_Ext()
   LIN {X -4.398, Y -11.255, Z 75.650}
   LaserEnd_Ext()
   LIN {X -4.398, Y 33.050, Z 75.650}
   LaserStart_Ext()
   LIN {X -4.398, Y 44.632, Z 75.650}
   LaserEnd_Ext()
   LIN {X -5.398, Y 44.360, Z 75.650}
   LaserStart_Ext()
   LIN {X -5.398, Y 36.009, Z 75.650}
   LaserEnd_Ext()
   LIN {X -5.398, Y -14.234, Z 75.650}
   LaserStart_Ext()
   LIN {X -5.398, Y -24.069, Z 75.650}
   LaserEnd_Ext()
   LIN {X -6.398, Y -21.892, Z 75.650}
   LaserStart_Ext()
   LIN {X -6.398, Y -17.209, Z 75.650}
   LaserEnd_Ext()
   LIN {X -6.398, Y 38.626, Z 75.650}
   LaserStart_Ext()
   LIN {X -6.398, Y 43.821, Z 75.650}
   LaserEnd_Ext()
   LIN {X -7.398, Y 41.782, Z 75.650}
   LaserStart_Ext()
   LIN {X -7.398, Y 41.371, Z 75.650}
   LaserEnd_Ext()
   LIN {X -3.142, Y -17.365, Z 76.500}
   LaserStart_Ext()
   LIN {X -3.011, Y -16.878, Z 76.500} C_DIS
   LIN {X -2.526, Y -16.374, Z 76.500} C_DIS
   LIN {X -1.552, Y -15.367, Z 76.500} C_DIS
   LIN {X -0.603, Y -14.998, Z 76.500} C_DIS
   LIN {X 0.476, Y -14.573, Z 76.500} C_DIS
   LIN {X 2.011, Y -14.661, Z 76.500} C_DIS
   LIN {X 2.631, Y -14.699, Z 76.500} C_DIS
   LIN {X 3.071, Y -14.938, Z 76.500} C_DIS
   LIN {X 4.500, Y -15.710, Z 76.500} C_DIS
   LIN {X 5.625, Y -17.343, Z 76.500} C_DIS
   LIN {X 5.941, Y -17.805, Z 76.500} C_DIS
   LIN {X 6.006, Y -18.361, Z 76.500} C_DIS
   LIN {X 6.203, Y -19.999, Z 76.500} C_DIS
   LIN {X 5.761, Y -21.242, Z 76.500} C_DIS
   LIN {X 5.397, Y -22.249, Z 76.500} C_DIS
   LIN {X 4.258, Y -23.382, Z 76.500} C_DIS
   LIN {X 3.921, Y -23.718, Z 76.500} C_DIS
   LIN {X 3.630, Y -23.826, Z 76.500} C_DIS
   LIN {X 1.849, Y -24.478, Z 76.500} C_DIS
   LIN {X 0.188, Y -24.361, Z 76.500} C_DIS
   LIN {X -0.194, Y -24.333, Z 76.500} C_DIS
   LIN {X -0.650, Y -24.087, Z 76.500} C_DIS
   LIN {X -2.015, Y -23.357, Z 76.500} C_DIS
   LIN {X -2.748, Y -22.418, Z 76.500} C_DIS
   LIN {X -3.295, Y -21.713, Z 76.500} C_DIS
   LIN {X -3.515, Y -20.783, Z 76.500} C_DIS
   LIN {X -3.780, Y -19.684, Z 76.500} C_DIS
   LIN {X -3.142, Y -17.365, Z 76.500}
   LaserEnd_Ext()
   LIN {X -8.172, Y 40.178, Z 76.500}
   LaserStart_Ext()
   LIN {X -7.953, Y 39.665, Z 76.500} C_DIS
   LIN {X -7.683, Y 39.026, Z 76.500} C_DIS
   LIN {X -7.108, Y 37.613, Z 76.500} C_DIS
   LIN {X -7.050, Y 37.466, Z 76.500} C_DIS
   LIN {X -6.246, Y 35.326, Z 76.500} C_DIS
   LIN {X -5.436, Y 32.913, Z 76.500} C_DIS
   LIN {X -5.320, Y 32.566, Z 76.500} C_DIS
   LIN {X -5.294, Y 32.467, Z 76.500} C_DIS
   LIN {X -5.022, Y 31.452, Z 76.500} C_DIS
   LIN {X -4.751, Y 30.438, Z 76.500} C_DIS
   LIN {X -3.887, Y 27.347, Z 76.500} C_DIS
   LIN {X -3.543, Y 25.729, Z 76.500} C_DIS
   LIN {X -2.374, Y 18.133, Z 76.500} C_DIS
   LIN {X -2.322, Y 17.840, Z 76.500} C_DIS
   LIN {X -2.296, Y 17.454, Z 76.500} C_DIS
   LIN {X -2.156, Y 6.509, Z 76.500} C_DIS
   LIN {X -2.445, Y 2.465, Z 76.500} C_DIS
   LIN {X -2.899, Y -0.549, Z 76.500} C_DIS
   LIN {X -3.595, Y -4.546, Z 76.500} C_DIS
   LIN {X -4.546, Y -8.413, Z 76.500} C_DIS
   LIN {X -4.683, Y -8.954, Z 76.500} C_DIS
   LIN {X -4.860, Y -9.528, Z 76.500} C_DIS
   LIN {X -5.781, Y -12.509, Z 76.500} C_DIS
   LIN {X -7.034, Y -15.920, Z 76.500} C_DIS
   LIN {X -7.149, Y -16.226, Z 76.500} C_DIS
   LIN {X -7.229, Y -16.606, Z 76.500} C_DIS
   LIN {X -7.790, Y -19.331, Z 76.500} C_DIS
   LIN {X -7.386, Y -21.521, Z 76.500} C_DIS
   LIN {X -7.127, Y -22.982, Z 76.500} C_DIS
   LIN {X -6.395, Y -24.179, Z 76.500} C_DIS
   LIN {X -5.599, Y -25.462, Z 76.500} C_DIS
   LIN {X -4.251, Y -26.564, Z 76.500} C_DIS
   LIN {X -3.238, Y -27.384, Z 76.500} C_DIS
   LIN {X -2.485, Y -27.716, Z 76.500} C_DIS
   LIN {X -1.260, Y -28.147, Z 76.500} C_DIS
   LIN {X 0.624, Y -28.395, Z 76.500} C_DIS
   LIN {X 1.520, Y -28.526, Z 76.500} C_DIS
   LIN {X 1.904, Y -28.456, Z 76.500} C_DIS
   LIN {X 4.170, Y -28.017, Z 76.500} C_DIS
   LIN {X 6.330, Y -26.645, Z 76.500} C_DIS
   LIN {X 7.529, Y -25.916, Z 76.500} C_DIS
   LIN {X 8.771, Y -24.195, Z 76.500} C_DIS
   LIN {X 9.315, Y -23.436, Z 76.500} C_DIS
   LIN {X 9.496, Y -22.844, Z 76.500} C_DIS
   LIN {X 10.170, Y -20.599, Z 76.500} C_DIS
   LIN {X 10.470, Y -17.952, Z 76.500} C_DIS
   LIN {X 10.534, Y -17.357, Z 76.500} C_DIS
   LIN {X 10.581, Y -16.760, Z 76.500} C_DIS
   LIN {X 10.783, Y -14.406, Z 76.500} C_DIS
   LIN {X 10.924, Y -11.904, Z 76.500} C_DIS
   LIN {X 10.987, Y -10.606, Z 76.500} C_DIS
   LIN {X 11.010, Y -8.642, Z 76.500} C_DIS
   LIN {X 11.058, Y -5.819, Z 76.500} C_DIS
   LIN {X 10.958, Y -2.763, Z 76.500} C_DIS
   LIN {X 10.821, Y 0.692, Z 76.500} C_DIS
   LIN {X 10.741, Y 1.992, Z 76.500} C_DIS
   LIN {X 10.407, Y 4.948, Z 76.500} C_DIS
   LIN {X 9.693, Y 10.555, Z 76.500} C_DIS
   LIN {X 8.455, Y 16.263, Z 76.500} C_DIS
   LIN {X 7.523, Y 21.091, Z 76.500} C_DIS
   LIN {X 7.053, Y 22.877, Z 76.500} C_DIS
   LIN {X 6.424, Y 24.843, Z 76.500} C_DIS
   LIN {X 4.618, Y 30.609, Z 76.500} C_DIS
   LIN {X 3.014, Y 34.797, Z 76.500} C_DIS
   LIN {X 2.756, Y 35.409, Z 76.500} C_DIS
   LIN {X 1.863, Y 37.543, Z 76.500} C_DIS
   LIN {X 0.942, Y 39.592, Z 76.500} C_DIS
   LIN {X 0.545, Y 40.459, Z 76.500} C_DIS
   LIN {X -0.197, Y 42.007, Z 76.500} C_DIS
   LIN {X -0.305, Y 42.231, Z 76.500} C_DIS
   LIN {X -0.392, Y 42.404, Z 76.500} C_DIS
   LIN {X -0.972, Y 43.567, Z 76.500} C_DIS
   LIN {X -1.622, Y 44.418, Z 76.500} C_DIS
   LIN {X -1.866, Y 44.735, Z 76.500} C_DIS
   LIN {X -2.572, Y 45.134, Z 76.500} C_DIS
   LIN {X -3.380, Y 45.593, Z 76.500} C_DIS
   LIN {X -3.848, Y 45.630, Z 76.500} C_DIS
   LIN {X -5.119, Y 45.726, Z 76.500} C_DIS
   LIN {X -7.330, Y 44.544, Z 76.500} C_DIS
   LIN {X -7.493, Y 44.458, Z 76.500} C_DIS
   LIN {X -7.548, Y 44.365, Z 76.500} C_DIS
   LIN {X -8.351, Y 42.941, Z 76.500} C_DIS
   LIN {X -8.475, Y 41.926, Z 76.500} C_DIS
   LIN {X -8.511, Y 41.558, Z 76.500} C_DIS
   LIN {X -8.397, Y 41.106, Z 76.500} C_DIS
   LIN {X -8.172, Y 40.178, Z 76.500}
   LaserEnd_Ext()
   LIN {X -3.519, Y 44.522, Z 76.500}
   LaserStart_Ext()
   LIN {X -5.252, Y 44.522, Z 76.500}
   LaserEnd_Ext()
   LIN {X -6.875, Y 43.522, Z 76.500}
   LaserStart_Ext()
   LIN {X -2.196, Y 43.522, Z 76.500}
   LaserEnd_Ext()
   LIN {X -1.568, Y 42.522, Z 76.500}
   LaserStart_Ext()
   LIN {X -7.395, Y 42.522, Z 76.500}
   LaserEnd_Ext()
   LIN {X -7.470, Y 41.522, Z 76.500}
   LaserStart_Ext()
   LIN {X -1.074, Y 41.522, Z 76.500}
   LaserEnd_Ext()
   LIN {X -0.594, Y 40.522, Z 76.500}
   LaserStart_Ext()
   LIN {X -7.227, Y 40.522, Z 76.500}
   LaserEnd_Ext()
   LIN {X -6.807, Y 39.522, Z 76.500}
   LaserStart_Ext()
   LIN {X -0.126, Y 39.522, Z 76.500}
   LaserEnd_Ext()
   LIN {X 0.326, Y 38.522, Z 76.500}
   LaserStart_Ext()
   LIN {X -6.398, Y 38.522, Z 76.500}
   LaserEnd_Ext()
   LIN {X -6.003, Y 37.522, Z 76.500}
   LaserStart_Ext()
   LIN {X 0.776, Y 37.522, Z 76.500}
   LaserEnd_Ext()
   LIN {X 1.206, Y 36.522, Z 76.500}
   LaserStart_Ext()
   LIN {X -5.627, Y 36.522, Z 76.500}
   LaserEnd_Ext()
   LIN {X -5.256, Y 35.522, Z 76.500}
   LaserStart_Ext()
   LIN {X 1.625, Y 35.522, Z 76.500}
   LaserEnd_Ext()
   LIN {X 2.045, Y 34.522, Z 76.500}
   LaserStart_Ext()
   LIN {X -4.921, Y 34.522, Z 76.500}
   LaserEnd_Ext()
   LIN {X -4.585, Y 33.522, Z 76.500}
   LaserStart_Ext()
   LIN {X 2.432, Y 33.522, Z 76.500}
   LaserEnd_Ext()
   LIN {X 2.815, Y 32.522, Z 76.500}
   LaserStart_Ext()
   LIN {X -4.273, Y 32.522, Z 76.500}
   LaserEnd_Ext()
   LIN {X -4.006, Y 31.522, Z 76.500}
   LaserStart_Ext()
   LIN {X 3.198, Y 31.522, Z 76.500}
   LaserEnd_Ext()
   LIN {X 3.581, Y 30.522, Z 76.500}
   LaserStart_Ext()
   LIN {X -3.736, Y 30.522, Z 76.500}
   LaserEnd_Ext()
   LIN {X -3.456, Y 29.522, Z 76.500}
   LaserStart_Ext()
   LIN {X 3.911, Y 29.522, Z 76.500}
   LaserEnd_Ext()
   LIN {X 4.224, Y 28.522, Z 76.500}
   LaserStart_Ext()
   LIN {X -3.177, Y 28.522, Z 76.500}
   LaserEnd_Ext()
   LIN {X -2.902, Y 27.522, Z 76.500}
   LaserStart_Ext()
   LIN {X 4.537, Y 27.522, Z 76.500}
   LaserEnd_Ext()
   LIN {X 4.850, Y 26.522, Z 76.500}
   LaserStart_Ext()
   LIN {X -2.689, Y 26.522, Z 76.500}
   LaserEnd_Ext()
   LIN {X -2.499, Y 25.522, Z 76.500}
   LaserStart_Ext()
   LIN {X 5.164, Y 25.522, Z 76.500}
   LaserEnd_Ext()
   LIN {X 5.477, Y 24.522, Z 76.500}
   LaserStart_Ext()
   LIN {X -2.345, Y 24.522, Z 76.500}
   LaserEnd_Ext()
   LIN {X -2.191, Y 23.522, Z 76.500}
   LaserStart_Ext()
   LIN {X 5.797, Y 23.522, Z 76.500}
   LaserEnd_Ext()
   LIN {X 6.112, Y 22.522, Z 76.500}
   LaserStart_Ext()
   LIN {X -2.037, Y 22.522, Z 76.500}
   LaserEnd_Ext()
   LIN {X -1.883, Y 21.522, Z 76.500}
   LaserStart_Ext()
   LIN {X 6.376, Y 21.522, Z 76.500}
   LaserEnd_Ext()
   LIN {X 6.614, Y 20.522, Z 76.500}
   LaserStart_Ext()
   LIN {X -1.729, Y 20.522, Z 76.500}
   LaserEnd_Ext()
   LIN {X -1.576, Y 19.522, Z 76.500}
   LaserStart_Ext()
   LIN {X 6.807, Y 19.522, Z 76.500}
   LaserEnd_Ext()
   LIN {X 7.000, Y 18.522, Z 76.500}
   LaserStart_Ext()
   LIN {X -1.422, Y 18.522, Z 76.500}
   LaserEnd_Ext()
   LIN {X -1.298, Y 17.522, Z 76.500}
   LaserStart_Ext()
   LIN {X 7.193, Y 17.522, Z 76.500}
   LaserEnd_Ext()
   LIN {X 7.386, Y 16.522, Z 76.500}
   LaserStart_Ext()
   LIN {X -1.284, Y 16.522, Z 76.500}
   LaserEnd_Ext()
   LIN {X -1.271, Y 15.522, Z 76.500}
   LaserStart_Ext()
   LIN {X 7.592, Y 15.522, Z 76.500}
   LaserEnd_Ext()
   LIN {X 7.809, Y 14.522, Z 76.500}
   LaserStart_Ext()
   LIN {X -1.258, Y 14.522, Z 76.500}
   LaserEnd_Ext()
   LIN {X -1.246, Y 13.522, Z 76.500}
   LaserStart_Ext()
   LIN {X 8.026, Y 13.522, Z 76.500}
   LaserEnd_Ext()
   LIN {X 8.243, Y 12.522, Z 76.500}
   LaserStart_Ext()
   LIN {X -1.233, Y 12.522, Z 76.500}
   LaserEnd_Ext()
   LIN {X -1.220, Y 11.522, Z 76.500}
   LaserStart_Ext()
   LIN {X 8.460, Y 11.522, Z 76.500}
   LaserEnd_Ext()
   LIN {X 8.677, Y 10.522, Z 76.500}
   LaserStart_Ext()
   LIN {X -1.207, Y 10.522, Z 76.500}
   LaserEnd_Ext()
   LIN {X -1.195, Y 9.522, Z 76.500}
   LaserStart_Ext()
   LIN {X 8.816, Y 9.522, Z 76.500}
   LaserEnd_Ext()
   LIN {X 8.944, Y 8.522, Z 76.500}
   LaserStart_Ext()
   LIN {X -1.182, Y 8.522, Z 76.500}
   LaserEnd_Ext()
   LIN {X -1.169, Y 7.522, Z 76.500}
   LaserStart_Ext()
   LIN {X 9.071, Y 7.522, Z 76.500}
   LaserEnd_Ext()
   LIN {X 9.199, Y 6.522, Z 76.500}
   LaserStart_Ext()
   LIN {X -1.157, Y 6.522, Z 76.500}
   LaserEnd_Ext()
   LIN {X -1.224, Y 5.522, Z 76.500}
   LaserStart_Ext()
   LIN {X 9.326, Y 5.522, Z 76.500}
   LaserEnd_Ext()
   LIN {X 9.449, Y 4.522, Z 76.500}
   LaserStart_Ext()
   LIN {X -1.296, Y 4.522, Z 76.500}
   LaserEnd_Ext()
   LIN {X -1.367, Y 3.522, Z 76.500}
   LaserStart_Ext()
   LIN {X 9.562, Y 3.522, Z 76.500}
   LaserEnd_Ext()
   LIN {X 9.675, Y 2.522, Z 76.500}
   LaserStart_Ext()
   LIN {X -1.438, Y 2.522, Z 76.500}
   LaserEnd_Ext()
   LIN {X -1.576, Y 1.522, Z 76.500}
   LaserStart_Ext()
   LIN {X 9.768, Y 1.522, Z 76.500}
   LaserEnd_Ext()
   LIN {X 9.827, Y 0.522, Z 76.500}
   LaserStart_Ext()
   LIN {X -1.726, Y 0.522, Z 76.500}
   LaserEnd_Ext()
   LIN {X -1.877, Y -0.478, Z 76.500}
   LaserStart_Ext()
   LIN {X 9.867, Y -0.478, Z 76.500}
   LaserEnd_Ext()
   LIN {X 9.906, Y -1.478, Z 76.500}
   LaserStart_Ext()
   LIN {X -2.046, Y -1.478, Z 76.500}
   LaserEnd_Ext()
   LIN {X -2.220, Y -2.478, Z 76.500}
   LaserStart_Ext()
   LIN {X 9.946, Y -2.478, Z 76.500}
   LaserEnd_Ext()
   LIN {X 9.981, Y -3.478, Z 76.500}
   LaserStart_Ext()
   LIN {X -2.394, Y -3.478, Z 76.500}
   LaserEnd_Ext()
   LIN {X -2.568, Y -4.478, Z 76.500}
   LaserStart_Ext()
   LIN {X 10.014, Y -4.478, Z 76.500}
   LaserEnd_Ext()
   LIN {X 10.046, Y -5.478, Z 76.500}
   LaserStart_Ext()
   LIN {X -2.795, Y -5.478, Z 76.500}
   LaserEnd_Ext()
   LIN {X -3.041, Y -6.478, Z 76.500}
   LaserStart_Ext()
   LIN {X 10.046, Y -6.478, Z 76.500}
   LaserEnd_Ext()
   LIN {X 10.029, Y -7.478, Z 76.500}
   LaserStart_Ext()
   LIN {X -3.286, Y -7.478, Z 76.500}
   LaserEnd_Ext()
   LIN {X -3.532, Y -8.478, Z 76.500}
   LaserStart_Ext()
   LIN {X 10.012, Y -8.478, Z 76.500}
   LaserEnd_Ext()
   LIN {X 10.000, Y -9.478, Z 76.500}
   LaserStart_Ext()
   LIN {X -3.798, Y -9.478, Z 76.500}
   LaserEnd_Ext()
   LIN {X -4.107, Y -10.478, Z 76.500}
   LaserStart_Ext()
   LIN {X 9.989, Y -10.478, Z 76.500}
   LaserEnd_Ext()
   LIN {X 9.943, Y -11.478, Z 76.500}
   LaserStart_Ext()
   LIN {X -4.416, Y -11.478, Z 76.500}
   LaserEnd_Ext()
   LIN {X -4.725, Y -12.478, Z 76.500}
   LaserStart_Ext()
   LIN {X 9.890, Y -12.478, Z 76.500}
   LaserEnd_Ext()
   LIN {X 9.834, Y -13.478, Z 76.500}
   LaserStart_Ext()
   LIN {X -5.072, Y -13.478, Z 76.500}
   LaserEnd_Ext()
   LIN {X -5.439, Y -14.478, Z 76.500}
   LaserStart_Ext()
   LIN {X -2.010, Y -14.478, Z 76.500}
   LaserEnd_Ext()
   LIN {X 4.324, Y -14.478, Z 76.500}
   LaserStart_Ext()
   LIN {X 9.773, Y -14.478, Z 76.500}
   LaserEnd_Ext()
   LIN {X 9.688, Y -15.478, Z 76.500}
   LaserStart_Ext()
   LIN {X 5.555, Y -15.478, Z 76.500}
   LaserEnd_Ext()
   LIN {X -3.051, Y -15.478, Z 76.500}
   LaserStart_Ext()
   LIN {X -5.806, Y -15.478, Z 76.500}
   LaserEnd_Ext()
   LIN {X -6.175, Y -16.478, Z 76.500}
   LaserStart_Ext()
   LIN {X -3.926, Y -16.478, Z 76.500}
   LaserEnd_Ext()
   LIN {X 6.244, Y -16.478, Z 76.500}
   LaserStart_Ext()
   LIN {X 9.602, Y -16.478, Z 76.500}
   LaserEnd_Ext()
   LIN {X 9.515, Y -17.478, Z 76.500}
   LaserStart_Ext()
   LIN {X 6.886, Y -17.478, Z 76.500}
   LaserEnd_Ext()
   LIN {X -4.211, Y -17.478, Z 76.500}
   LaserStart_Ext()
   LIN {X -6.387, Y -17.478, Z 76.500}
   LaserEnd_Ext()
   LIN {X -6.593, Y -18.478, Z 76.500}
   LaserStart_Ext()
   LIN {X -4.486, Y -18.478, Z 76.500}
   LaserEnd_Ext()
   LIN {X 7.028, Y -18.478, Z 76.500}
   LaserStart_Ext()
   LIN {X 9.404, Y -18.478, Z 76.500}
   LaserEnd_Ext()
   LIN {X 9.290, Y -19.478, Z 76.500}
   LaserStart_Ext()
   LIN {X 7.148, Y -19.478, Z 76.500}
   LaserEnd_Ext()
   LIN {X -4.757, Y -19.478, Z 76.500}
   LaserStart_Ext()
   LIN {X -6.746, Y -19.478, Z 76.500}
   LaserEnd_Ext()
   LIN {X -6.562, Y -20.478, Z 76.500}
   LaserStart_Ext()
   LIN {X -4.617, Y -20.478, Z 76.500}
   LaserEnd_Ext()
   LIN {X 7.094, Y -20.478, Z 76.500}
   LaserStart_Ext()
   LIN {X 9.162, Y -20.478, Z 76.500}
   LaserEnd_Ext()
   LIN {X 8.862, Y -21.478, Z 76.500}
   LaserStart_Ext()
   LIN {X 6.739, Y -21.478, Z 76.500}
   LaserEnd_Ext()
   LIN {X -4.378, Y -21.478, Z 76.500}
   LaserStart_Ext()
   LIN {X -6.378, Y -21.478, Z 76.500}
   LaserEnd_Ext()
   LIN {X -6.200, Y -22.478, Z 76.500}
   LaserStart_Ext()
   LIN {X -3.967, Y -22.478, Z 76.500}
   LaserEnd_Ext()
   LIN {X 6.378, Y -22.478, Z 76.500}
   LaserStart_Ext()
   LIN {X 8.562, Y -22.478, Z 76.500}
   LaserEnd_Ext()
   LIN {X 8.054, Y -23.478, Z 76.500}
   LaserStart_Ext()
   LIN {X 5.579, Y -23.478, Z 76.500}
   LaserEnd_Ext()
   LIN {X -3.189, Y -23.478, Z 76.500}
   LaserStart_Ext()
   LIN {X -5.651, Y -23.478, Z 76.500}
   LaserEnd_Ext()
   LIN {X -5.033, Y -24.478, Z 76.500}
   LaserStart_Ext()
   LIN {X -2.038, Y -24.478, Z 76.500}
   LaserEnd_Ext()
   LIN {X 4.569, Y -24.478, Z 76.500}
   LaserStart_Ext()
   LIN {X 7.333, Y -24.478, Z 76.500}
   LaserEnd_Ext()
   LIN {X 6.324, Y -25.478, Z 76.500}
   LaserStart_Ext()
   LIN {X -3.999, Y -25.478, Z 76.500}
   LaserEnd_Ext()
   LIN {X -2.767, Y -26.478, Z 76.500}
   LaserStart_Ext()
   LIN {X 4.727, Y -26.478, Z 76.500}
   LaserEnd_Ext()
   LIN {X 1.689, Y -27.478, Z 76.500}
   LaserStart_Ext()
   LIN {X 1.270, Y -27.478, Z 76.500}
   LaserEnd_Ext()
   LIN {X 5.630, Y -21.771, Z 77.350}
   LaserStart_Ext()
   LIN {X 5.485, Y -22.183, Z 77.350} C_DIS
   LIN {X 5.326, Y -22.342, Z 77.350} C_DIS
   LIN {X 4.011, Y -23.657, Z 77.350} C_DIS
   LIN {X 2.514, Y -24.212, Z 77.350} C_DIS
   LIN {X 1.941, Y -24.422, Z 77.350} C_DIS
   LIN {X 1.117, Y -24.364, Z 77.350} C_DIS
   LIN {X -0.102, Y -24.281, Z 77.350} C_DIS
   LIN {X -0.880, Y -23.869, Z 77.350} C_DIS
   LIN {X -1.926, Y -23.309, Z 77.350} C_DIS
   LIN {X -2.874, Y -22.096, Z 77.350} C_DIS
   LIN {X -3.210, Y -21.669, Z 77.350} C_DIS
   LIN {X -3.341, Y -21.131, Z 77.350} C_DIS
   LIN {X -3.700, Y -19.641, Z 77.350} C_DIS
   LIN {X -3.394, Y -18.528, Z 77.350} C_DIS
   LIN {X -2.936, Y -16.831, Z 77.350} C_DIS
   LIN {X -1.639, Y -15.484, Z 77.350} C_DIS
   LIN {X -1.480, Y -15.317, Z 77.350} C_DIS
   LIN {X -1.165, Y -15.192, Z 77.350} C_DIS
   LIN {X 0.541, Y -14.521, Z 77.350} C_DIS
   LIN {X 1.888, Y -14.598, Z 77.350} C_DIS
   LIN {X 2.699, Y -14.640, Z 77.350} C_DIS
   LIN {X 3.550, Y -15.096, Z 77.350} C_DIS
   LIN {X 4.570, Y -15.647, Z 77.350} C_DIS
   LIN {X 5.341, Y -16.764, Z 77.350} C_DIS
   LIN {X 6.017, Y -17.739, Z 77.350} C_DIS
   LIN {X 6.137, Y -18.711, Z 77.350} C_DIS
   LIN {X 6.284, Y -19.933, Z 77.350} C_DIS
   LIN {X 5.630, Y -21.771, Z 77.350}
   LaserEnd_Ext()
   LIN {X -7.608, Y 38.737, Z 77.350}
   LaserStart_Ext()
   LIN {X -7.741, Y 39.060, Z 77.350} C_DIS
   LIN {X -7.911, Y 39.456, Z 77.350} C_DIS
   LIN {X -8.233, Y 40.210, Z 77.350} C_DIS
   LIN {X -8.374, Y 40.796, Z 77.350} C_DIS
   LIN {X -8.577, Y 41.621, Z 77.350} C_DIS
   LIN {X -8.448, Y 42.645, Z 77.350} C_DIS
   LIN {X -8.402, Y 43.024, Z 77.350} C_DIS
   LIN {X -8.235, Y 43.321, Z 77.350} C_DIS
   LIN {X -7.528, Y 44.531, Z 77.350} C_DIS
   LIN {X -5.387, Y 45.662, Z 77.350} C_DIS
   LIN {X -5.193, Y 45.766, Z 77.350} C_DIS
   LIN {X -4.970, Y 45.749, Z 77.350} C_DIS
   LIN {X -3.452, Y 45.636, Z 77.350} C_DIS
   LIN {X -2.617, Y 45.167, Z 77.350} C_DIS
   LIN {X -1.937, Y 44.782, Z 77.350} C_DIS
   LIN {X -1.286, Y 43.935, Z 77.350} C_DIS
   LIN {X -1.040, Y 43.616, Z 77.350} C_DIS
   LIN {X -0.912, Y 43.363, Z 77.350} C_DIS
   LIN {X -0.369, Y 42.278, Z 77.350} C_DIS
   LIN {X 0.363, Y 40.760, Z 77.350} C_DIS
   LIN {X 0.507, Y 40.464, Z 77.350} C_DIS
   LIN {X 1.323, Y 38.679, Z 77.350} C_DIS
   LIN {X 1.818, Y 37.577, Z 77.350} C_DIS
   LIN {X 2.298, Y 36.431, Z 77.350} C_DIS
   LIN {X 3.057, Y 34.629, Z 77.350} C_DIS
   LIN {X 3.128, Y 34.460, Z 77.350} C_DIS
   LIN {X 4.616, Y 30.576, Z 77.350} C_DIS
   LIN {X 6.769, Y 23.702, Z 77.350} C_DIS
   LIN {X 7.179, Y 22.421, Z 77.350} C_DIS
   LIN {X 7.485, Y 21.257, Z 77.350} C_DIS
   LIN {X 8.092, Y 18.111, Z 77.350} C_DIS
   LIN {X 9.654, Y 10.912, Z 77.350} C_DIS
   LIN {X 10.554, Y 3.840, Z 77.350} C_DIS
   LIN {X 10.795, Y 1.707, Z 77.350} C_DIS
   LIN {X 10.853, Y 0.770, Z 77.350} C_DIS
   LIN {X 11.074, Y -4.791, Z 77.350} C_DIS
   LIN {X 11.105, Y -5.741, Z 77.350} C_DIS
   LIN {X 11.090, Y -6.618, Z 77.350} C_DIS
   LIN {X 11.046, Y -10.528, Z 77.350} C_DIS
   LIN {X 10.919, Y -13.111, Z 77.350} C_DIS
   LIN {X 10.851, Y -14.328, Z 77.350} C_DIS
   LIN {X 10.753, Y -15.474, Z 77.350} C_DIS
   LIN {X 10.608, Y -17.279, Z 77.350} C_DIS
   LIN {X 10.416, Y -19.080, Z 77.350} C_DIS
   LIN {X 10.252, Y -20.523, Z 77.350} C_DIS
   LIN {X 9.651, Y -22.527, Z 77.350} C_DIS
   LIN {X 9.380, Y -23.409, Z 77.350} C_DIS
   LIN {X 9.070, Y -23.818, Z 77.350} C_DIS
   LIN {X 7.565, Y -25.903, Z 77.350} C_DIS
   LIN {X 5.269, Y -27.299, Z 77.350} C_DIS
   LIN {X 4.193, Y -27.982, Z 77.350} C_DIS
   LIN {X 2.622, Y -28.287, Z 77.350} C_DIS
   LIN {X 1.552, Y -28.471, Z 77.350} C_DIS
   LIN {X -0.699, Y -28.176, Z 77.350} C_DIS
   LIN {X -3.067, Y -27.343, Z 77.350} C_DIS
   LIN {X -3.201, Y -27.306, Z 77.350} C_DIS
   LIN {X -3.314, Y -27.215, Z 77.350} C_DIS
   LIN {X -5.506, Y -25.423, Z 77.350} C_DIS
   LIN {X -6.942, Y -23.105, Z 77.350} C_DIS
   LIN {X -7.039, Y -22.947, Z 77.350} C_DIS
   LIN {X -7.074, Y -22.754, Z 77.350} C_DIS
   LIN {X -7.711, Y -19.297, Z 77.350} C_DIS
   LIN {X -7.248, Y -17.048, Z 77.350} C_DIS
   LIN {X -7.077, Y -16.191, Z 77.350} C_DIS
   LIN {X -6.573, Y -14.799, Z 77.350} C_DIS
   LIN {X -5.716, Y -12.463, Z 77.350} C_DIS
   LIN {X -5.198, Y -10.790, Z 77.350} C_DIS
   LIN {X -4.685, Y -9.118, Z 77.350} C_DIS
   LIN {X -4.287, Y -7.547, Z 77.350} C_DIS
   LIN {X -3.639, Y -4.913, Z 77.350} C_DIS
   LIN {X -2.755, Y 0.162, Z 77.350} C_DIS
   LIN {X -2.466, Y 2.082, Z 77.350} C_DIS
   LIN {X -2.115, Y 7.000, Z 77.350} C_DIS
   LIN {X -2.231, Y 16.077, Z 77.350} C_DIS
   LIN {X -2.373, Y 18.187, Z 77.350} C_DIS
   LIN {X -2.655, Y 19.785, Z 77.350} C_DIS
   LIN {X -3.595, Y 25.895, Z 77.350} C_DIS
   LIN {X -3.873, Y 27.197, Z 77.350} C_DIS
   LIN {X -4.888, Y 30.833, Z 77.350} C_DIS
   LIN {X -5.208, Y 32.026, Z 77.350} C_DIS
   LIN {X -5.363, Y 32.605, Z 77.350} C_DIS
   LIN {X -6.270, Y 35.293, Z 77.350} C_DIS
   LIN {X -6.320, Y 35.430, Z 77.350} C_DIS
   LIN {X -7.134, Y 37.580, Z 77.350} C_DIS
   LIN {X -7.608, Y 38.737, Z 77.350}
   LaserEnd_Ext()
   LIN {X -7.280, Y 40.525, Z 77.350}
   LaserStart_Ext()
   LIN {X -7.280, Y 42.973, Z 77.350}
   LaserEnd_Ext()
   LIN {X -6.280, Y 44.059, Z 77.350}
   LaserStart_Ext()
   LIN {X -6.280, Y 38.133, Z 77.350}
   LaserEnd_Ext()
   LIN {X -6.280, Y -17.306, Z 77.350}
   LaserStart_Ext()
   LIN {X -6.280, Y -21.544, Z 77.350}
   LaserEnd_Ext()
   LIN {X -5.280, Y -23.890, Z 77.350}
   LaserStart_Ext()
   LIN {X -5.280, Y -14.177, Z 77.350}
   LaserEnd_Ext()
   LIN {X -5.280, Y 35.485, Z 77.350}
   LaserStart_Ext()
   LIN {X -5.280, Y 44.588, Z 77.350}
   LaserEnd_Ext()
   LIN {X -4.280, Y 44.695, Z 77.350}
   LaserStart_Ext()
   LIN {X -4.280, Y 32.428, Z 77.350}
   LaserEnd_Ext()
   LIN {X -4.280, Y -11.204, Z 77.350}
   LaserStart_Ext()
   LIN {X -4.280, Y -17.973, Z 77.350}
   LaserEnd_Ext()
   LIN {X -4.280, Y -21.503, Z 77.350}
   LaserStart_Ext()
   LIN {X -4.280, Y -25.134, Z 77.350}
   LaserEnd_Ext()
   LIN {X -3.280, Y -25.951, Z 77.350}
   LaserStart_Ext()
   LIN {X -3.280, Y -23.201, Z 77.350}
   LaserEnd_Ext()
   LIN {X -3.280, Y -15.746, Z 77.350}
   LaserStart_Ext()
   LIN {X -3.280, Y -7.641, Z 77.350}
   LaserEnd_Ext()
   LIN {X -3.280, Y 28.792, Z 77.350}
   LaserStart_Ext()
   LIN {X -3.280, Y 44.392, Z 77.350}
   LaserEnd_Ext()
   LIN {X -2.280, Y 43.587, Z 77.350}
   LaserStart_Ext()
   LIN {X -2.280, Y 23.922, Z 77.350}
   LaserEnd_Ext()
   LIN {X -2.280, Y -2.938, Z 77.350}
   LaserStart_Ext()
   LIN {X -2.280, Y -14.707, Z 77.350}
   LaserEnd_Ext()
   LIN {X -2.280, Y -24.254, Z 77.350}
   LaserStart_Ext()
   LIN {X -2.280, Y -26.559, Z 77.350}
   LaserEnd_Ext()
   LIN {X -1.280, Y -26.911, Z 77.350}
   LaserStart_Ext()
   LIN {X -1.280, Y -24.789, Z 77.350}
   LaserEnd_Ext()
   LIN {X -1.280, Y -14.163, Z 77.350}
   LaserStart_Ext()
   LIN {X -1.280, Y 4.651, Z 77.350}
   LaserEnd_Ext()
   LIN {X -1.280, Y 16.839, Z 77.350}
   LaserStart_Ext()
   LIN {X -1.280, Y 41.865, Z 77.350}
   LaserEnd_Ext()
   LIN {X -0.280, Y 39.780, Z 77.350}
   LaserStart_Ext()
   LIN {X -0.280, Y -13.769, Z 77.350}
   LaserEnd_Ext()
   LIN {X -0.280, Y -25.265, Z 77.350}
   LaserStart_Ext()
   LIN {X -0.280, Y -27.222, Z 77.350}
   LaserEnd_Ext()
   LIN {X 0.720, Y -27.353, Z 77.350}
   LaserStart_Ext()
   LIN {X 0.720, Y -25.339, Z 77.350}
   LaserEnd_Ext()
   LIN {X 0.720, Y -13.530, Z 77.350}
   LaserStart_Ext()
   LIN {X 0.720, Y 37.581, Z 77.350}
   LaserEnd_Ext()
   LIN {X 1.720, Y 35.227, Z 77.350}
   LaserStart_Ext()
   LIN {X 1.720, Y -13.587, Z 77.350}
   LaserEnd_Ext()
   LIN {X 1.720, Y -25.409, Z 77.350}
   LaserStart_Ext()
   LIN {X 1.720, Y -27.427, Z 77.350}
   LaserEnd_Ext()
   LIN {X 2.720, Y -27.249, Z 77.350}
   LaserStart_Ext()
   LIN {X 2.720, Y -25.201, Z 77.350}
   LaserEnd_Ext()
   LIN {X 2.720, Y -13.640, Z 77.350}
   LaserStart_Ext()
   LIN {X 2.720, Y 32.729, Z 77.350}
   LaserEnd_Ext()
   LIN {X 3.720, Y 30.090, Z 77.350}
   LaserStart_Ext()
   LIN {X 3.720, Y -14.053, Z 77.350}
   LaserEnd_Ext()
   LIN {X 3.720, Y -24.831, Z 77.350}
   LaserStart_Ext()
   LIN {X 3.720, Y -27.055, Z 77.350}
   LaserEnd_Ext()
   LIN {X 4.720, Y -26.463, Z 77.350}
   LaserStart_Ext()
   LIN {X 4.720, Y -24.362, Z 77.350}
   LaserEnd_Ext()
   LIN {X 4.720, Y -14.592, Z 77.350}
   LaserStart_Ext()
   LIN {X 4.720, Y 26.897, Z 77.350}
   LaserEnd_Ext()
   LIN {X 5.720, Y 23.705, Z 77.350}
   LaserStart_Ext()
   LIN {X 5.720, Y -15.553, Z 77.350}
   LaserEnd_Ext()
   LIN {X 5.720, Y -23.362, Z 77.350}
   LaserStart_Ext()
   LIN {X 5.720, Y -25.854, Z 77.350}
   LaserEnd_Ext()
   LIN {X 6.720, Y -25.247, Z 77.350}
   LaserStart_Ext()
   LIN {X 6.720, Y -21.691, Z 77.350}
   LaserEnd_Ext()
   LIN {X 6.720, Y -16.998, Z 77.350}
   LaserStart_Ext()
   LIN {X 6.720, Y 19.943, Z 77.350}
   LaserEnd_Ext()
   LIN {X 7.720, Y 15.109, Z 77.350}
   LaserStart_Ext()
   LIN {X 7.720, Y -23.980, Z 77.350}
   LaserEnd_Ext()
   LIN {X 8.720, Y -22.149, Z 77.350}
   LaserStart_Ext()
   LIN {X 8.720, Y 10.326, Z 77.350}
   LaserEnd_Ext()
   LIN {X 9.720, Y 2.317, Z 77.350}
   LaserStart_Ext()
   LIN {X 9.720, Y -15.839, Z 77.350}
   LaserEnd_Ext()
   LIN {X 5.569, Y -22.120, Z 78.200}
   LaserStart_Ext()
   LIN {X 4.556, Y -23.141, Z 78.200} C_DIS
   LIN {X 4.101, Y -23.595, Z 78.200} C_DIS
   LIN {X 3.063, Y -23.980, Z 78.200} C_DIS
   LIN {X 2.033, Y -24.365, Z 78.200} C_DIS
   LIN {X 1.385, Y -24.324, Z 78.200} C_DIS
   LIN {X -0.011, Y -24.230, Z 78.200} C_DIS
   LIN {X -1.757, Y -23.305, Z 78.200} C_DIS
   LIN {X -1.885, Y -23.202, Z 78.200} C_DIS
   LIN {X -3.125, Y -21.625, Z 78.200} C_DIS
   LIN {X -3.594, Y -19.705, Z 78.200} C_DIS
   LIN {X -3.620, Y -19.598, Z 78.200} C_DIS
   LIN {X -3.531, Y -19.265, Z 78.200} C_DIS
   LIN {X -2.862, Y -16.785, Z 78.200} C_DIS
   LIN {X -2.390, Y -16.295, Z 78.200} C_DIS
   LIN {X -1.408, Y -15.267, Z 78.200} C_DIS
   LIN {X 0.532, Y -14.497, Z 78.200} C_DIS
   LIN {X 0.662, Y -14.472, Z 78.200} C_DIS
   LIN {X 2.767, Y -14.582, Z 78.200} C_DIS
   LIN {X 4.349, Y -15.430, Z 78.200} C_DIS
   LIN {X 4.641, Y -15.585, Z 78.200} C_DIS
   LIN {X 4.894, Y -15.947, Z 78.200} C_DIS
   LIN {X 6.093, Y -17.672, Z 78.200} C_DIS
   LIN {X 6.329, Y -19.584, Z 78.200} C_DIS
   LIN {X 6.365, Y -19.866, Z 78.200} C_DIS
   LIN {X 6.286, Y -20.093, Z 78.200} C_DIS
   LIN {X 5.569, Y -22.120, Z 78.200}
   LaserEnd_Ext()
   LIN {X 10.334, Y -20.447, Z 78.200}
   LaserStart_Ext()
   LIN {X 10.235, Y -20.778, Z 78.200} C_DIS
   LIN {X 9.420, Y -23.430, Z 78.200} C_DIS
   LIN {X 8.489, Y -24.660, Z 78.200} C_DIS
   LIN {X 7.602, Y -25.890, Z 78.200} C_DIS
   LIN {X 4.233, Y -27.937, Z 78.200} C_DIS
   LIN {X 1.491, Y -28.418, Z 78.200} C_DIS
   LIN {X -0.137, Y -28.204, Z 78.200} C_DIS
   LIN {X -1.850, Y -27.602, Z 78.200} C_DIS
   LIN {X -3.103, Y -27.261, Z 78.200} C_DIS
   LIN {X -4.158, Y -26.410, Z 78.200} C_DIS
   LIN {X -5.412, Y -25.384, Z 78.200} C_DIS
   LIN {X -6.352, Y -23.869, Z 78.200} C_DIS
   LIN {X -6.951, Y -22.911, Z 78.200} C_DIS
   LIN {X -7.268, Y -21.236, Z 78.200} C_DIS
   LIN {X -7.632, Y -19.264, Z 78.200} C_DIS
   LIN {X -7.401, Y -18.141, Z 78.200} C_DIS
   LIN {X -7.005, Y -16.156, Z 78.200} C_DIS
   LIN {X -5.838, Y -12.930, Z 78.200} C_DIS
   LIN {X -5.651, Y -12.418, Z 78.200} C_DIS
   LIN {X -5.537, Y -12.051, Z 78.200} C_DIS
   LIN {X -4.687, Y -9.283, Z 78.200} C_DIS
   LIN {X -4.027, Y -6.681, Z 78.200} C_DIS
   LIN {X -3.683, Y -5.280, Z 78.200} C_DIS
   LIN {X -2.611, Y 0.874, Z 78.200} C_DIS
   LIN {X -2.486, Y 1.699, Z 78.200} C_DIS
   LIN {X -2.073, Y 7.492, Z 78.200} C_DIS
   LIN {X -2.165, Y 14.700, Z 78.200} C_DIS
   LIN {X -2.425, Y 18.535, Z 78.200} C_DIS
   LIN {X -2.936, Y 21.437, Z 78.200} C_DIS
   LIN {X -3.648, Y 26.062, Z 78.200} C_DIS
   LIN {X -3.858, Y 27.046, Z 78.200} C_DIS
   LIN {X -5.026, Y 31.229, Z 78.200} C_DIS
   LIN {X -5.393, Y 32.601, Z 78.200} C_DIS
   LIN {X -5.473, Y 32.847, Z 78.200} C_DIS
   LIN {X -6.343, Y 35.400, Z 78.200} C_DIS
   LIN {X -7.110, Y 37.412, Z 78.200} C_DIS
   LIN {X -7.188, Y 37.615, Z 78.200} C_DIS
   LIN {X -7.260, Y 37.789, Z 78.200} C_DIS
   LIN {X -7.798, Y 39.093, Z 78.200} C_DIS
   LIN {X -8.080, Y 39.751, Z 78.200} C_DIS
   LIN {X -8.293, Y 40.242, Z 78.200} C_DIS
   LIN {X -8.505, Y 41.096, Z 78.200} C_DIS
   LIN {X -8.640, Y 41.645, Z 78.200} C_DIS
   LIN {X -8.585, Y 42.085, Z 78.200} C_DIS
   LIN {X -8.454, Y 43.100, Z 78.200} C_DIS
   LIN {X -7.671, Y 44.418, Z 78.200} C_DIS
   LIN {X -7.563, Y 44.603, Z 78.200} C_DIS
   LIN {X -7.323, Y 44.730, Z 78.200} C_DIS
   LIN {X -5.266, Y 45.805, Z 78.200} C_DIS
   LIN {X -4.026, Y 45.717, Z 78.200} C_DIS
   LIN {X -3.525, Y 45.680, Z 78.200} C_DIS
   LIN {X -2.857, Y 45.304, Z 78.200} C_DIS
   LIN {X -2.008, Y 44.829, Z 78.200} C_DIS
   LIN {X -1.626, Y 44.337, Z 78.200} C_DIS
   LIN {X -1.108, Y 43.665, Z 78.200} C_DIS
   LIN {X -0.548, Y 42.556, Z 78.200} C_DIS
   LIN {X -0.432, Y 42.327, Z 78.200} C_DIS
   LIN {X -0.270, Y 41.994, Z 78.200} C_DIS
   LIN {X 0.469, Y 40.469, Z 78.200} C_DIS
   LIN {X 1.705, Y 37.765, Z 78.200} C_DIS
   LIN {X 1.774, Y 37.612, Z 78.200} C_DIS
   LIN {X 1.840, Y 37.452, Z 78.200} C_DIS
   LIN {X 3.123, Y 34.409, Z 78.200} C_DIS
   LIN {X 3.242, Y 34.123, Z 78.200} C_DIS
   LIN {X 4.613, Y 30.544, Z 78.200} C_DIS
   LIN {X 7.114, Y 22.560, Z 78.200} C_DIS
   LIN {X 7.305, Y 21.964, Z 78.200} C_DIS
   LIN {X 7.447, Y 21.423, Z 78.200} C_DIS
   LIN {X 7.730, Y 19.959, Z 78.200} C_DIS
   LIN {X 9.614, Y 11.269, Z 78.200} C_DIS
   LIN {X 10.702, Y 2.733, Z 78.200} C_DIS
   LIN {X 10.850, Y 1.423, Z 78.200} C_DIS
   LIN {X 10.885, Y 0.847, Z 78.200} C_DIS
   LIN {X 11.078, Y -3.993, Z 78.200} C_DIS
   LIN {X 11.153, Y -5.663, Z 78.200} C_DIS
   LIN {X 11.149, Y -6.566, Z 78.200} C_DIS
   LIN {X 11.105, Y -10.450, Z 78.200} C_DIS
   LIN {X 10.922, Y -14.168, Z 78.200} C_DIS
   LIN {X 10.914, Y -14.317, Z 78.200} C_DIS
   LIN {X 10.683, Y -17.202, Z 78.200} C_DIS
   LIN {X 10.361, Y -20.209, Z 78.200} C_DIS
   LIN {X 10.334, Y -20.447, Z 78.200}
   LaserEnd_Ext()
   LIN {X 1.117, Y -27.360, Z 78.200}
   LaserStart_Ext()
   LIN {X 1.739, Y -27.360, Z 78.200}
   LaserEnd_Ext()
   LIN {X 4.903, Y -26.360, Z 78.200}
   LaserStart_Ext()
   LIN {X -2.606, Y -26.360, Z 78.200}
   LaserEnd_Ext()
   LIN {X -3.862, Y -25.360, Z 78.200}
   LaserStart_Ext()
   LIN {X 1.919, Y -25.360, Z 78.200}
   LaserEnd_Ext()
   LIN {X 2.120, Y -25.360, Z 78.200}
   LaserStart_Ext()
   LIN {X 6.548, Y -25.360, Z 78.200}
   LaserEnd_Ext()
   LIN {X 7.473, Y -24.360, Z 78.200}
   LaserStart_Ext()
   LIN {X 4.744, Y -24.360, Z 78.200}
   LaserEnd_Ext()
   LIN {X -1.901, Y -24.360, Z 78.200}
   LaserStart_Ext()
   LIN {X -4.871, Y -24.360, Z 78.200}
   LaserEnd_Ext()
   LIN {X -5.491, Y -23.360, Z 78.200}
   LaserStart_Ext()
   LIN {X -3.033, Y -23.360, Z 78.200}
   LaserEnd_Ext()
   LIN {X 5.747, Y -23.360, Z 78.200}
   LaserStart_Ext()
   LIN {X 8.219, Y -23.360, Z 78.200}
   LaserEnd_Ext()
   LIN {X 8.702, Y -22.360, Z 78.200}
   LaserStart_Ext()
   LIN {X 6.545, Y -22.360, Z 78.200}
   LaserEnd_Ext()
   LIN {X -3.819, Y -22.360, Z 78.200}
   LaserStart_Ext()
   LIN {X -6.038, Y -22.360, Z 78.200}
   LaserEnd_Ext()
   LIN {X -6.227, Y -21.360, Z 78.200}
   LaserStart_Ext()
   LIN {X -4.219, Y -21.360, Z 78.200}
   LaserEnd_Ext()
   LIN {X 6.899, Y -21.360, Z 78.200}
   LaserStart_Ext()
   LIN {X 9.010, Y -21.360, Z 78.200}
   LaserEnd_Ext()
   LIN {X 9.316, Y -20.360, Z 78.200}
   LaserStart_Ext()
   LIN {X 7.252, Y -20.360, Z 78.200}
   LaserEnd_Ext()
   LIN {X -4.463, Y -20.360, Z 78.200}
   LaserStart_Ext()
   LIN {X -6.413, Y -20.360, Z 78.200}
   LaserEnd_Ext()
   LIN {X -6.598, Y -19.360, Z 78.200}
   LaserStart_Ext()
   LIN {X -4.590, Y -19.360, Z 78.200}
   LaserEnd_Ext()
   LIN {X 7.309, Y -19.360, Z 78.200}
   LaserStart_Ext()
   LIN {X 9.446, Y -19.360, Z 78.200}
   LaserEnd_Ext()
   LIN {X 9.553, Y -18.360, Z 78.200}
   LaserStart_Ext()
   LIN {X 7.186, Y -18.360, Z 78.200}
   LaserEnd_Ext()
   LIN {X -4.322, Y -18.360, Z 78.200}
   LaserStart_Ext()
   LIN {X -6.425, Y -18.360, Z 78.200}
   LaserEnd_Ext()
   LIN {X -6.225, Y -17.360, Z 78.200}
   LaserStart_Ext()
   LIN {X -4.053, Y -17.360, Z 78.200}
   LaserEnd_Ext()
   LIN {X 7.043, Y -17.360, Z 78.200}
   LaserStart_Ext()
   LIN {X 9.660, Y -17.360, Z 78.200}
   LaserEnd_Ext()
   LIN {X 9.747, Y -16.360, Z 78.200}
   LaserStart_Ext()
   LIN {X 6.399, Y -16.360, Z 78.200}
   LaserEnd_Ext()
   LIN {X -3.766, Y -16.360, Z 78.200}
   LaserStart_Ext()
   LIN {X -6.015, Y -16.360, Z 78.200}
   LaserEnd_Ext()
   LIN {X -5.654, Y -15.360, Z 78.200}
   LaserStart_Ext()
   LIN {X -2.880, Y -15.360, Z 78.200}
   LaserEnd_Ext()
   LIN {X 5.704, Y -15.360, Z 78.200}
   LaserStart_Ext()
   LIN {X 9.827, Y -15.360, Z 78.200}
   LaserEnd_Ext()
   LIN {X 9.907, Y -14.360, Z 78.200}
   LaserStart_Ext()
   LIN {X 4.470, Y -14.360, Z 78.200}
   LaserEnd_Ext()
   LIN {X -1.825, Y -14.360, Z 78.200}
   LaserStart_Ext()
   LIN {X -5.292, Y -14.360, Z 78.200}
   LaserEnd_Ext()
   LIN {X -4.931, Y -13.360, Z 78.200}
   LaserStart_Ext()
   LIN {X 9.961, Y -13.360, Z 78.200}
   LaserEnd_Ext()
   LIN {X 10.010, Y -12.360, Z 78.200}
   LaserStart_Ext()
   LIN {X -4.586, Y -12.360, Z 78.200}
   LaserEnd_Ext()
   LIN {X -4.279, Y -11.360, Z 78.200}
   LaserStart_Ext()
   LIN {X 10.059, Y -11.360, Z 78.200}
   LaserEnd_Ext()
   LIN {X 10.106, Y -10.360, Z 78.200}
   LaserStart_Ext()
   LIN {X -3.972, Y -10.360, Z 78.200}
   LaserEnd_Ext()
   LIN {X -3.675, Y -9.360, Z 78.200}
   LaserStart_Ext()
   LIN {X 10.117, Y -9.360, Z 78.200}
   LaserEnd_Ext()
   LIN {X 10.128, Y -8.360, Z 78.200}
   LaserStart_Ext()
   LIN {X -3.421, Y -8.360, Z 78.200}
   LaserEnd_Ext()
   LIN {X -3.168, Y -7.360, Z 78.200}
   LaserStart_Ext()
   LIN {X 10.140, Y -7.360, Z 78.200}
   LaserEnd_Ext()
   LIN {X 10.150, Y -6.360, Z 78.200}
   LaserStart_Ext()
   LIN {X -2.918, Y -6.360, Z 78.200}
   LaserEnd_Ext()
   LIN {X -2.682, Y -5.360, Z 78.200}
   LaserStart_Ext()
   LIN {X 10.138, Y -5.360, Z 78.200}
   LaserEnd_Ext()
   LIN {X 10.093, Y -4.360, Z 78.200}
   LaserStart_Ext()
   LIN {X -2.507, Y -4.360, Z 78.200}
   LaserEnd_Ext()
   LIN {X -2.333, Y -3.360, Z 78.200}
   LaserStart_Ext()
   LIN {X 10.052, Y -3.360, Z 78.200}
   LaserEnd_Ext()
   LIN {X 10.012, Y -2.360, Z 78.200}
   LaserStart_Ext()
   LIN {X -2.159, Y -2.360, Z 78.200}
   LaserEnd_Ext()
   LIN {X -1.985, Y -1.360, Z 78.200}
   LaserStart_Ext()
   LIN {X 9.972, Y -1.360, Z 78.200}
   LaserEnd_Ext()
   LIN {X 9.932, Y -0.360, Z 78.200}
   LaserStart_Ext()
   LIN {X -1.811, Y -0.360, Z 78.200}
   LaserEnd_Ext()
   LIN {X -1.637, Y 0.640, Z 78.200}
   LaserStart_Ext()
   LIN {X 9.893, Y 0.640, Z 78.200}
   LaserEnd_Ext()
   LIN {X 9.819, Y 1.640, Z 78.200}
   LaserStart_Ext()
   LIN {X -1.488, Y 1.640, Z 78.200}
   LaserEnd_Ext()
   LIN {X -1.417, Y 2.640, Z 78.200}
   LaserStart_Ext()
   LIN {X 9.706, Y 2.640, Z 78.200}
   LaserEnd_Ext()
   LIN {X 9.578, Y 3.640, Z 78.200}
   LaserStart_Ext()
   LIN {X -1.345, Y 3.640, Z 78.200}
   LaserEnd_Ext()
   LIN {X -1.274, Y 4.640, Z 78.200}
   LaserStart_Ext()
   LIN {X 9.451, Y 4.640, Z 78.200}
   LaserEnd_Ext()
   LIN {X 9.323, Y 5.640, Z 78.200}
   LaserStart_Ext()
   LIN {X -1.203, Y 5.640, Z 78.200}
   LaserEnd_Ext()
   LIN {X -1.132, Y 6.640, Z 78.200}
   LaserStart_Ext()
   LIN {X 9.196, Y 6.640, Z 78.200}
   LaserEnd_Ext()
   LIN {X 9.069, Y 7.640, Z 78.200}
   LaserStart_Ext()
   LIN {X -1.075, Y 7.640, Z 78.200}
   LaserEnd_Ext()
   LIN {X -1.088, Y 8.640, Z 78.200}
   LaserStart_Ext()
   LIN {X 8.941, Y 8.640, Z 78.200}
   LaserEnd_Ext()
   LIN {X 8.814, Y 9.640, Z 78.200}
   LaserStart_Ext()
   LIN {X -1.101, Y 9.640, Z 78.200}
   LaserEnd_Ext()
   LIN {X -1.113, Y 10.640, Z 78.200}
   LaserStart_Ext()
   LIN {X 8.686, Y 10.640, Z 78.200}
   LaserEnd_Ext()
   LIN {X 8.511, Y 11.640, Z 78.200}
   LaserStart_Ext()
   LIN {X -1.126, Y 11.640, Z 78.200}
   LaserEnd_Ext()
   LIN {X -1.139, Y 12.640, Z 78.200}
   LaserStart_Ext()
   LIN {X 8.294, Y 12.640, Z 78.200}
   LaserEnd_Ext()
   LIN {X 8.077, Y 13.640, Z 78.200}
   LaserStart_Ext()
   LIN {X -1.152, Y 13.640, Z 78.200}
   LaserEnd_Ext()
   LIN {X -1.164, Y 14.640, Z 78.200}
   LaserStart_Ext()
   LIN {X 7.860, Y 14.640, Z 78.200}
   LaserEnd_Ext()
   LIN {X 7.643, Y 15.640, Z 78.200}
   LaserStart_Ext()
   LIN {X -1.227, Y 15.640, Z 78.200}
   LaserEnd_Ext()
   LIN {X -1.294, Y 16.640, Z 78.200}
   LaserStart_Ext()
   LIN {X 7.426, Y 16.640, Z 78.200}
   LaserEnd_Ext()
   LIN {X 7.209, Y 17.640, Z 78.200}
   LaserStart_Ext()
   LIN {X -1.362, Y 17.640, Z 78.200}
   LaserEnd_Ext()
   LIN {X -1.432, Y 18.640, Z 78.200}
   LaserStart_Ext()
   LIN {X 6.993, Y 18.640, Z 78.200}
   LaserEnd_Ext()
   LIN {X 6.776, Y 19.640, Z 78.200}
   LaserStart_Ext()
   LIN {X -1.604, Y 19.640, Z 78.200}
   LaserEnd_Ext()
   LIN {X -1.780, Y 20.640, Z 78.200}
   LaserStart_Ext()
   LIN {X 6.580, Y 20.640, Z 78.200}
   LaserEnd_Ext()
   LIN {X 6.356, Y 21.640, Z 78.200}
   LaserStart_Ext()
   LIN {X -1.956, Y 21.640, Z 78.200}
   LaserEnd_Ext()
   LIN {X -2.110, Y 22.640, Z 78.200}
   LaserStart_Ext()
   LIN {X 6.041, Y 22.640, Z 78.200}
   LaserEnd_Ext()
   LIN {X 5.728, Y 23.640, Z 78.200}
   LaserStart_Ext()
   LIN {X -2.264, Y 23.640, Z 78.200}
   LaserEnd_Ext()
   LIN {X -2.417, Y 24.640, Z 78.200}
   LaserStart_Ext()
   LIN {X 5.415, Y 24.640, Z 78.200}
   LaserEnd_Ext()
   LIN {X 5.101, Y 25.640, Z 78.200}
   LaserStart_Ext()
   LIN {X -2.571, Y 25.640, Z 78.200}
   LaserEnd_Ext()
   LIN {X -2.749, Y 26.640, Z 78.200}
   LaserStart_Ext()
   LIN {X 4.788, Y 26.640, Z 78.200}
   LaserEnd_Ext()
   LIN {X 4.475, Y 27.640, Z 78.200}
   LaserStart_Ext()
   LIN {X -2.985, Y 27.640, Z 78.200}
   LaserEnd_Ext()
   LIN {X -3.265, Y 28.640, Z 78.200}
   LaserStart_Ext()
   LIN {X 4.162, Y 28.640, Z 78.200}
   LaserEnd_Ext()
   LIN {X 3.848, Y 29.640, Z 78.200}
   LaserStart_Ext()
   LIN {X -3.544, Y 29.640, Z 78.200}
   LaserEnd_Ext()
   LIN {X -3.823, Y 30.640, Z 78.200}
   LaserStart_Ext()
   LIN {X 3.506, Y 30.640, Z 78.200}
   LaserEnd_Ext()
   LIN {X 3.123, Y 31.640, Z 78.200}
   LaserStart_Ext()
   LIN {X -4.101, Y 31.640, Z 78.200}
   LaserEnd_Ext()
   LIN {X -4.368, Y 32.640, Z 78.200}
   LaserStart_Ext()
   LIN {X 2.740, Y 32.640, Z 78.200}
   LaserEnd_Ext()
   LIN {X 2.357, Y 33.640, Z 78.200}
   LaserStart_Ext()
   LIN {X -4.687, Y 33.640, Z 78.200}
   LaserEnd_Ext()
   LIN {X -5.028, Y 34.640, Z 78.200}
   LaserStart_Ext()
   LIN {X 1.940, Y 34.640, Z 78.200}
   LaserEnd_Ext()
   LIN {X 1.519, Y 35.640, Z 78.200}
   LaserStart_Ext()
   LIN {X -5.368, Y 35.640, Z 78.200}
   LaserEnd_Ext()
   LIN {X -5.746, Y 36.640, Z 78.200}
   LaserStart_Ext()
   LIN {X 1.098, Y 36.640, Z 78.200}
   LaserEnd_Ext()
   LIN {X 0.662, Y 37.640, Z 78.200}
   LaserStart_Ext()
   LIN {X -6.127, Y 37.640, Z 78.200}
   LaserEnd_Ext()
   LIN {X -6.529, Y 38.640, Z 78.200}
   LaserStart_Ext()
   LIN {X 0.205, Y 38.640, Z 78.200}
   LaserEnd_Ext()
   LIN {X -0.252, Y 39.640, Z 78.200}
   LaserStart_Ext()
   LIN {X -6.944, Y 39.640, Z 78.200}
   LaserEnd_Ext()
   LIN {X -7.361, Y 40.640, Z 78.200}
   LaserStart_Ext()
   LIN {X -0.725, Y 40.640, Z 78.200}
   LaserEnd_Ext()
   LIN {X -1.210, Y 41.640, Z 78.200}
   LaserStart_Ext()
   LIN {X -7.609, Y 41.640, Z 78.200}
   LaserEnd_Ext()
   LIN {X -7.505, Y 42.640, Z 78.200}
   LaserStart_Ext()
   LIN {X -1.711, Y 42.640, Z 78.200}
   LaserEnd_Ext()
   LIN {X -2.351, Y 43.640, Z 78.200}
   LaserStart_Ext()
   LIN {X -6.970, Y 43.640, Z 78.200}
   LaserEnd_Ext()
   LIN {X -5.337, Y 44.640, Z 78.200}
   LaserStart_Ext()
   LIN {X -3.716, Y 44.640, Z 78.200}
   LaserEnd_Ext()
   LIN {X -2.702, Y -22.011, Z 79.050}
   LaserStart_Ext()
   LIN {X -3.040, Y -21.580, Z 79.050} C_DIS
   LIN {X -3.168, Y -21.057, Z 79.050} C_DIS
   LIN {X -3.540, Y -19.555, Z 79.050} C_DIS
   LIN {X -2.942, Y -17.325, Z 79.050} C_DIS
   LIN {X -2.786, Y -16.735, Z 79.050} C_DIS
   LIN {X -2.272, Y -16.197, Z 79.050} C_DIS
   LIN {X -1.336, Y -15.218, Z 79.050} C_DIS
   LIN {X -0.432, Y -14.859, Z 79.050} C_DIS
   LIN {X 0.681, Y -14.414, Z 79.050} C_DIS
   LIN {X 2.270, Y -14.494, Z 79.050} C_DIS
   LIN {X 2.836, Y -14.524, Z 79.050} C_DIS
   LIN {X 3.236, Y -14.738, Z 79.050} C_DIS
   LIN {X 4.712, Y -15.522, Z 79.050} C_DIS
   LIN {X 5.990, Y -17.350, Z 79.050} C_DIS
   LIN {X 6.169, Y -17.606, Z 79.050} C_DIS
   LIN {X 6.204, Y -17.891, Z 79.050} C_DIS
   LIN {X 6.446, Y -19.799, Z 79.050} C_DIS
   LIN {X 5.907, Y -21.341, Z 79.050} C_DIS
   LIN {X 5.654, Y -22.057, Z 79.050} C_DIS
   LIN {X 4.867, Y -22.850, Z 79.050} C_DIS
   LIN {X 4.190, Y -23.534, Z 79.050} C_DIS
   LIN {X 3.624, Y -23.748, Z 79.050} C_DIS
   LIN {X 2.124, Y -24.309, Z 79.050} C_DIS
   LIN {X 0.244, Y -24.189, Z 79.050} C_DIS
   LIN {X 0.080, Y -24.178, Z 79.050} C_DIS
   LIN {X -0.126, Y -24.069, Z 79.050} C_DIS
   LIN {X -1.749, Y -23.215, Z 79.050} C_DIS
   LIN {X -2.702, Y -22.011, Z 79.050}
   LaserEnd_Ext()
   LIN {X -2.079, Y 44.876, Z 79.050}
   LaserStart_Ext()
   LIN {X -1.535, Y 44.175, Z 79.050} C_DIS
   LIN {X -1.176, Y 43.714, Z 79.050} C_DIS
   LIN {X -0.963, Y 43.296, Z 79.050} C_DIS
   LIN {X -0.501, Y 42.385, Z 79.050} C_DIS
   LIN {X 0.118, Y 41.114, Z 79.050} C_DIS
   LIN {X 0.421, Y 40.495, Z 79.050} C_DIS
   LIN {X 0.814, Y 39.643, Z 79.050} C_DIS
   LIN {X 1.739, Y 37.623, Z 79.050} C_DIS
   LIN {X 2.449, Y 35.939, Z 79.050} C_DIS
   LIN {X 3.190, Y 34.189, Z 79.050} C_DIS
   LIN {X 3.240, Y 34.065, Z 79.050} C_DIS
   LIN {X 3.356, Y 33.786, Z 79.050} C_DIS
   LIN {X 4.611, Y 30.511, Z 79.050} C_DIS
   LIN {X 7.380, Y 21.669, Z 79.050} C_DIS
   LIN {X 7.414, Y 21.571, Z 79.050} C_DIS
   LIN {X 7.470, Y 21.331, Z 79.050} C_DIS
   LIN {X 9.575, Y 11.626, Z 79.050} C_DIS
   LIN {X 10.849, Y 1.625, Z 79.050} C_DIS
   LIN {X 10.904, Y 1.138, Z 79.050} C_DIS
   LIN {X 10.917, Y 0.924, Z 79.050} C_DIS
   LIN {X 10.989, Y -0.874, Z 79.050} C_DIS
   LIN {X 11.200, Y -5.584, Z 79.050} C_DIS
   LIN {X 11.189, Y -8.133, Z 79.050} C_DIS
   LIN {X 11.164, Y -10.372, Z 79.050} C_DIS
   LIN {X 11.058, Y -12.515, Z 79.050} C_DIS
   LIN {X 10.986, Y -14.173, Z 79.050} C_DIS
   LIN {X 10.888, Y -15.489, Z 79.050} C_DIS
   LIN {X 10.757, Y -17.125, Z 79.050} C_DIS
   LIN {X 10.542, Y -19.137, Z 79.050} C_DIS
   LIN {X 10.417, Y -20.371, Z 79.050} C_DIS
   LIN {X 10.170, Y -21.140, Z 79.050} C_DIS
   LIN {X 9.460, Y -23.451, Z 79.050} C_DIS
   LIN {X 7.909, Y -25.503, Z 79.050} C_DIS
   LIN {X 7.638, Y -25.877, Z 79.050} C_DIS
   LIN {X 6.612, Y -26.501, Z 79.050} C_DIS
   LIN {X 4.499, Y -27.813, Z 79.050} C_DIS
   LIN {X 3.107, Y -28.075, Z 79.050} C_DIS
   LIN {X 1.429, Y -28.364, Z 79.050} C_DIS
   LIN {X 0.424, Y -28.233, Z 79.050} C_DIS
   LIN {X -0.634, Y -27.860, Z 79.050} C_DIS
   LIN {X -3.006, Y -27.216, Z 79.050} C_DIS
   LIN {X -5.002, Y -25.605, Z 79.050} C_DIS
   LIN {X -5.319, Y -25.346, Z 79.050} C_DIS
   LIN {X -5.556, Y -24.963, Z 79.050} C_DIS
   LIN {X -6.864, Y -22.876, Z 79.050} C_DIS
   LIN {X -7.552, Y -19.234, Z 79.050} C_DIS
   LIN {X -6.933, Y -16.121, Z 79.050} C_DIS
   LIN {X -5.943, Y -13.382, Z 79.050} C_DIS
   LIN {X -5.612, Y -12.458, Z 79.050} C_DIS
   LIN {X -5.396, Y -11.749, Z 79.050} C_DIS
   LIN {X -4.689, Y -9.448, Z 79.050} C_DIS
   LIN {X -3.767, Y -5.814, Z 79.050} C_DIS
   LIN {X -3.726, Y -5.647, Z 79.050} C_DIS
   LIN {X -3.296, Y -3.174, Z 79.050} C_DIS
   LIN {X -2.555, Y 1.048, Z 79.050} C_DIS
   LIN {X -2.514, Y 1.282, Z 79.050} C_DIS
   LIN {X -2.491, Y 1.466, Z 79.050} C_DIS
   LIN {X -2.455, Y 2.043, Z 79.050} C_DIS
   LIN {X -2.032, Y 7.983, Z 79.050} C_DIS
   LIN {X -2.100, Y 13.323, Z 79.050} C_DIS
   LIN {X -2.476, Y 18.882, Z 79.050} C_DIS
   LIN {X -3.217, Y 23.088, Z 79.050} C_DIS
   LIN {X -3.701, Y 26.228, Z 79.050} C_DIS
   LIN {X -3.843, Y 26.896, Z 79.050} C_DIS
   LIN {X -5.164, Y 31.624, Z 79.050} C_DIS
   LIN {X -5.447, Y 32.683, Z 79.050} C_DIS
   LIN {X -6.318, Y 35.225, Z 79.050} C_DIS
   LIN {X -6.392, Y 35.436, Z 79.050} C_DIS
   LIN {X -6.470, Y 35.638, Z 79.050} C_DIS
   LIN {X -7.241, Y 37.649, Z 79.050} C_DIS
   LIN {X -7.691, Y 38.733, Z 79.050} C_DIS
   LIN {X -7.855, Y 39.126, Z 79.050} C_DIS
   LIN {X -8.065, Y 39.608, Z 79.050} C_DIS
   LIN {X -8.353, Y 40.274, Z 79.050} C_DIS
   LIN {X -8.489, Y 40.820, Z 79.050} C_DIS
   LIN {X -8.704, Y 41.704, Z 79.050} C_DIS
   LIN {X -8.551, Y 42.836, Z 79.050} C_DIS
   LIN {X -8.507, Y 43.174, Z 79.050} C_DIS
   LIN {X -8.344, Y 43.448, Z 79.050} C_DIS
   LIN {X -7.659, Y 44.608, Z 79.050} C_DIS
   LIN {X -5.906, Y 45.548, Z 79.050} C_DIS
   LIN {X -5.338, Y 45.844, Z 79.050} C_DIS
   LIN {X -4.786, Y 45.805, Z 79.050} C_DIS
   LIN {X -3.598, Y 45.723, Z 79.050} C_DIS
   LIN {X -2.790, Y 45.274, Z 79.050} C_DIS
   LIN {X -2.079, Y 44.876, Z 79.050}
   LaserEnd_Ext()
   LIN {X 9.602, Y -18.526, Z 79.050}
   LaserStart_Ext()
   LIN {X 9.602, Y 3.503, Z 79.050}
   LaserEnd_Ext()
   LIN {X 8.602, Y 11.352, Z 79.050}
   LaserStart_Ext()
   LIN {X 8.602, Y -22.839, Z 79.050}
   LaserEnd_Ext()
   LIN {X 7.602, Y -24.250, Z 79.050}
   LaserStart_Ext()
   LIN {X 7.602, Y 16.006, Z 79.050}
   LaserEnd_Ext()
   LIN {X 6.602, Y 20.617, Z 79.050}
   LaserStart_Ext()
   LIN {X 6.602, Y -16.479, Z 79.050}
   LaserEnd_Ext()
   LIN {X 6.602, Y -22.377, Z 79.050}
   LaserStart_Ext()
   LIN {X 6.602, Y -25.337, Z 79.050}
   LaserEnd_Ext()
   LIN {X 5.602, Y -25.951, Z 79.050}
   LaserStart_Ext()
   LIN {X 5.602, Y -23.529, Z 79.050}
   LaserEnd_Ext()
   LIN {X 5.602, Y -15.050, Z 79.050}
   LaserStart_Ext()
   LIN {X 5.602, Y 24.002, Z 79.050}
   LaserEnd_Ext()
   LIN {X 4.602, Y 27.194, Z 79.050}
   LaserStart_Ext()
   LIN {X 4.602, Y -14.331, Z 79.050}
   LaserEnd_Ext()
   LIN {X 4.602, Y -24.444, Z 79.050}
   LaserStart_Ext()
   LIN {X 4.602, Y -26.572, Z 79.050}
   LaserEnd_Ext()
   LIN {X 3.602, Y -26.964, Z 79.050}
   LaserStart_Ext()
   LIN {X 3.602, Y -24.824, Z 79.050}
   LaserEnd_Ext()
   LIN {X 3.602, Y -13.800, Z 79.050}
   LaserStart_Ext()
   LIN {X 3.602, Y 30.349, Z 79.050}
   LaserEnd_Ext()
   LIN {X 2.602, Y 32.960, Z 79.050}
   LaserStart_Ext()
   LIN {X 2.602, Y -13.510, Z 79.050}
   LaserEnd_Ext()
   LIN {X 2.602, Y -25.198, Z 79.050}
   LaserStart_Ext()
   LIN {X 2.602, Y -27.147, Z 79.050}
   LaserEnd_Ext()
   LIN {X 1.602, Y -27.320, Z 79.050}
   LaserStart_Ext()
   LIN {X 1.602, Y -25.277, Z 79.050}
   LaserEnd_Ext()
   LIN {X 1.602, Y -13.459, Z 79.050}
   LaserStart_Ext()
   LIN {X 1.602, Y 35.375, Z 79.050}
   LaserEnd_Ext()
   LIN {X 0.602, Y 37.705, Z 79.050}
   LaserStart_Ext()
   LIN {X 0.602, Y -13.418, Z 79.050}
   LaserEnd_Ext()
   LIN {X 0.602, Y -25.214, Z 79.050}
   LaserStart_Ext()
   LIN {X 0.602, Y -27.235, Z 79.050}
   LaserEnd_Ext()
   LIN {X -0.398, Y -26.888, Z 79.050}
   LaserStart_Ext()
   LIN {X -0.398, Y -25.056, Z 79.050}
   LaserEnd_Ext()
   LIN {X -0.398, Y -13.768, Z 79.050}
   LaserStart_Ext()
   LIN {X -0.398, Y 39.883, Z 79.050}
   LaserEnd_Ext()
   LIN {X -1.398, Y 41.942, Z 79.050}
   LaserStart_Ext()
   LIN {X -1.398, Y 17.764, Z 79.050}
   LaserEnd_Ext()
   LIN {X -1.398, Y 2.811, Z 79.050}
   LaserStart_Ext()
   LIN {X -1.398, Y -14.166, Z 79.050}
   LaserEnd_Ext()
   LIN {X -1.398, Y -24.529, Z 79.050}
   LaserStart_Ext()
   LIN {X -1.398, Y -26.617, Z 79.050}
   LaserEnd_Ext()
   LIN {X -2.398, Y -26.345, Z 79.050}
   LaserStart_Ext()
   LIN {X -2.398, Y -23.974, Z 79.050}
   LaserEnd_Ext()
   LIN {X -2.398, Y -14.882, Z 79.050}
   LaserStart_Ext()
   LIN {X -2.398, Y -3.849, Z 79.050}
   LaserEnd_Ext()
   LIN {X -2.398, Y 24.338, Z 79.050}
   LaserStart_Ext()
   LIN {X -2.398, Y 43.656, Z 79.050}
   LaserEnd_Ext()
   LIN {X -3.398, Y 44.468, Z 79.050}
   LaserStart_Ext()
   LIN {X -3.398, Y 29.020, Z 79.050}
   LaserEnd_Ext()
   LIN {X -3.398, Y -8.425, Z 79.050}
   LaserStart_Ext()
   LIN {X -3.398, Y -15.929, Z 79.050}
   LaserEnd_Ext()
   LIN {X -3.398, Y -22.742, Z 79.050}
   LaserStart_Ext()
   LIN {X -3.398, Y -25.614, Z 79.050}
   LaserEnd_Ext()
   LIN {X -4.398, Y -24.807, Z 79.050}
   LaserStart_Ext()
   LIN {X -4.398, Y -20.249, Z 79.050}
   LaserEnd_Ext()
   LIN {X -4.398, Y -18.895, Z 79.050}
   LaserStart_Ext()
   LIN {X -4.398, Y -11.907, Z 79.050}
   LaserEnd_Ext()
   LIN {X -4.398, Y 32.632, Z 79.050}
   LaserStart_Ext()
   LIN {X -4.398, Y 44.776, Z 79.050}
   LaserEnd_Ext()
   LIN {X -5.398, Y 44.685, Z 79.050}
   LaserStart_Ext()
   LIN {X -5.398, Y 35.623, Z 79.050}
   LaserEnd_Ext()
   LIN {X -5.398, Y -14.817, Z 79.050}
   LaserStart_Ext()
   LIN {X -5.398, Y -23.332, Z 79.050}
   LaserEnd_Ext()
   LIN {X -6.398, Y -19.956, Z 79.050}
   LaserStart_Ext()
   LIN {X -6.398, Y -18.557, Z 79.050}
   LaserEnd_Ext()
   LIN {X -6.398, Y 38.226, Z 79.050}
   LaserStart_Ext()
   LIN {X -6.398, Y 44.149, Z 79.050}
   LaserEnd_Ext()
   LIN {X -7.398, Y 43.084, Z 79.050}
   LaserStart_Ext()
   LIN {X -7.398, Y 40.586, Z 79.050}
   LaserEnd_Ext()
   LIN {X 0.171, Y -24.126, Z 79.900}
   LaserStart_Ext()
   LIN {X -0.872, Y -23.582, Z 79.900} C_DIS
   LIN {X -1.660, Y -23.167, Z 79.900} C_DIS
   LIN {X -2.322, Y -22.331, Z 79.900} C_DIS
   LIN {X -2.955, Y -21.536, Z 79.900} C_DIS
   LIN {X -3.207, Y -20.531, Z 79.900} C_DIS
   LIN {X -3.460, Y -19.511, Z 79.900} C_DIS
   LIN {X -3.228, Y -18.647, Z 79.900} C_DIS
   LIN {X -2.708, Y -16.683, Z 79.900} C_DIS
   LIN {X -1.452, Y -15.366, Z 79.900} C_DIS
   LIN {X -1.263, Y -15.167, Z 79.900} C_DIS
   LIN {X 0.758, Y -14.359, Z 79.900} C_DIS
   LIN {X 2.023, Y -14.423, Z 79.900} C_DIS
   LIN {X 2.904, Y -14.465, Z 79.900} C_DIS
   LIN {X 3.900, Y -14.990, Z 79.900} C_DIS
   LIN {X 4.783, Y -15.459, Z 79.900} C_DIS
   LIN {X 5.389, Y -16.326, Z 79.900} C_DIS
   LIN {X 6.244, Y -17.540, Z 79.900} C_DIS
   LIN {X 6.391, Y -18.661, Z 79.900} C_DIS
   LIN {X 6.527, Y -19.732, Z 79.900} C_DIS
   LIN {X 6.026, Y -21.166, Z 79.900} C_DIS
   LIN {X 5.739, Y -21.994, Z 79.900} C_DIS
   LIN {X 5.354, Y -22.386, Z 79.900} C_DIS
   LIN {X 4.278, Y -23.474, Z 79.900} C_DIS
   LIN {X 2.510, Y -24.142, Z 79.900} C_DIS
   LIN {X 2.215, Y -24.252, Z 79.900} C_DIS
   LIN {X 1.766, Y -24.223, Z 79.900} C_DIS
   LIN {X 0.171, Y -24.126, Z 79.900}
   LaserEnd_Ext()
   LIN {X -5.509, Y 32.781, Z 79.900}
   LaserStart_Ext()
   LIN {X -6.440, Y 35.473, Z 79.900} C_DIS
   LIN {X -7.168, Y 37.357, Z 79.900} C_DIS
   LIN {X -7.295, Y 37.684, Z 79.900} C_DIS
   LIN {X -7.413, Y 37.964, Z 79.900} C_DIS
   LIN {X -7.912, Y 39.159, Z 79.900} C_DIS
   LIN {X -8.175, Y 39.763, Z 79.900} C_DIS
   LIN {X -8.413, Y 40.306, Z 79.900} C_DIS
   LIN {X -8.657, Y 41.318, Z 79.900} C_DIS
   LIN {X -8.770, Y 41.780, Z 79.900} C_DIS
   LIN {X -8.720, Y 42.148, Z 79.900} C_DIS
   LIN {X -8.583, Y 43.176, Z 79.900} C_DIS
   LIN {X -8.026, Y 44.158, Z 79.900} C_DIS
   LIN {X -7.762, Y 44.604, Z 79.900} C_DIS
   LIN {X -6.964, Y 45.033, Z 79.900} C_DIS
   LIN {X -5.411, Y 45.883, Z 79.900} C_DIS
   LIN {X -4.443, Y 45.819, Z 79.900} C_DIS
   LIN {X -3.671, Y 45.766, Z 79.900} C_DIS
   LIN {X -2.818, Y 45.292, Z 79.900} C_DIS
   LIN {X -2.149, Y 44.922, Z 79.900} C_DIS
   LIN {X -1.784, Y 44.456, Z 79.900} C_DIS
   LIN {X -1.244, Y 43.763, Z 79.900} C_DIS
   LIN {X -0.731, Y 42.757, Z 79.900} C_DIS
   LIN {X -0.551, Y 42.405, Z 79.900} C_DIS
   LIN {X -0.314, Y 41.923, Z 79.900} C_DIS
   LIN {X 0.357, Y 40.555, Z 79.900} C_DIS
   LIN {X 1.569, Y 37.928, Z 79.900} C_DIS
   LIN {X 1.709, Y 37.625, Z 79.900} C_DIS
   LIN {X 3.257, Y 33.968, Z 79.900} C_DIS
   LIN {X 3.365, Y 33.702, Z 79.900} C_DIS
   LIN {X 3.471, Y 33.449, Z 79.900} C_DIS
   LIN {X 4.608, Y 30.479, Z 79.900} C_DIS
   LIN {X 7.120, Y 22.459, Z 79.900} C_DIS
   LIN {X 7.409, Y 21.601, Z 79.900} C_DIS
   LIN {X 7.903, Y 19.511, Z 79.900} C_DIS
   LIN {X 9.536, Y 11.983, Z 79.900} C_DIS
   LIN {X 10.774, Y 2.264, Z 79.900} C_DIS
   LIN {X 10.949, Y 1.009, Z 79.900} C_DIS
   LIN {X 10.994, Y 0.141, Z 79.900} C_DIS
   LIN {X 11.248, Y -5.506, Z 79.900} C_DIS
   LIN {X 11.229, Y -9.701, Z 79.900} C_DIS
   LIN {X 11.222, Y -10.294, Z 79.900} C_DIS
   LIN {X 11.194, Y -10.861, Z 79.900} C_DIS
   LIN {X 11.054, Y -14.095, Z 79.900} C_DIS
   LIN {X 10.863, Y -16.661, Z 79.900} C_DIS
   LIN {X 10.832, Y -17.048, Z 79.900} C_DIS
   LIN {X 10.781, Y -17.524, Z 79.900} C_DIS
   LIN {X 10.499, Y -20.294, Z 79.900} C_DIS
   LIN {X 9.946, Y -22.022, Z 79.900} C_DIS
   LIN {X 9.500, Y -23.472, Z 79.900} C_DIS
   LIN {X 8.133, Y -25.280, Z 79.900} C_DIS
   LIN {X 7.674, Y -25.863, Z 79.900} C_DIS
   LIN {X 7.098, Y -26.240, Z 79.900} C_DIS
   LIN {X 4.781, Y -27.679, Z 79.900} C_DIS
   LIN {X 2.006, Y -28.201, Z 79.900} C_DIS
   LIN {X 1.368, Y -28.311, Z 79.900} C_DIS
   LIN {X 0.985, Y -28.261, Z 79.900} C_DIS
   LIN {X 0.583, Y -28.119, Z 79.900} C_DIS
   LIN {X -2.908, Y -27.172, Z 79.900} C_DIS
   LIN {X -4.565, Y -25.833, Z 79.900} C_DIS
   LIN {X -5.225, Y -25.306, Z 79.900} C_DIS
   LIN {X -5.657, Y -24.627, Z 79.900} C_DIS
   LIN {X -6.776, Y -22.840, Z 79.900} C_DIS
   LIN {X -7.213, Y -20.531, Z 79.900} C_DIS
   LIN {X -7.474, Y -19.196, Z 79.900} C_DIS
   LIN {X -7.165, Y -17.611, Z 79.900} C_DIS
   LIN {X -6.861, Y -16.085, Z 79.900} C_DIS
   LIN {X -6.374, Y -14.739, Z 79.900} C_DIS
   LIN {X -5.585, Y -12.531, Z 79.900} C_DIS
   LIN {X -5.067, Y -10.837, Z 79.900} C_DIS
   LIN {X -4.691, Y -9.613, Z 79.900} C_DIS
   LIN {X -4.147, Y -7.469, Z 79.900} C_DIS
   LIN {X -3.686, Y -5.635, Z 79.900} C_DIS
   LIN {X -2.772, Y -0.425, Z 79.900} C_DIS
   LIN {X -2.560, Y 0.762, Z 79.900} C_DIS
   LIN {X -2.494, Y 1.193, Z 79.900} C_DIS
   LIN {X -2.446, Y 1.694, Z 79.900} C_DIS
   LIN {X -2.266, Y 4.613, Z 79.900} C_DIS
   LIN {X -1.990, Y 8.475, Z 79.900} C_DIS
   LIN {X -2.035, Y 11.947, Z 79.900} C_DIS
   LIN {X -2.527, Y 19.229, Z 79.900} C_DIS
   LIN {X -3.499, Y 24.740, Z 79.900} C_DIS
   LIN {X -3.753, Y 26.394, Z 79.900} C_DIS
   LIN {X -3.828, Y 26.746, Z 79.900} C_DIS
   LIN {X -5.301, Y 32.020, Z 79.900} C_DIS
   LIN {X -5.486, Y 32.712, Z 79.900}
   LaserEnd_Ext()
   LIN {X -3.491, Y 44.522, Z 79.900}
   LaserStart_Ext()
   LIN {X -5.815, Y 44.522, Z 79.900}
   LaserEnd_Ext()
   LIN {X -7.237, Y 43.522, Z 79.900}
   LaserStart_Ext()
   LIN {X -2.324, Y 43.522, Z 79.900}
   LaserEnd_Ext()
   LIN {X -1.734, Y 42.522, Z 79.900}
   LaserStart_Ext()
   LIN {X -7.661, Y 42.522, Z 79.900}
   LaserEnd_Ext()
   LIN {X -7.677, Y 41.522, Z 79.900}
   LaserStart_Ext()
   LIN {X -1.231, Y 41.522, Z 79.900}
   LaserEnd_Ext()
   LIN {X -0.741, Y 40.522, Z 79.900}
   LaserStart_Ext()
   LIN {X -7.416, Y 40.522, Z 79.900}
   LaserEnd_Ext()
   LIN {X -6.980, Y 39.522, Z 79.900}
   LaserStart_Ext()
   LIN {X -0.268, Y 39.522, Z 79.900}
   LaserEnd_Ext()
   LIN {X 0.194, Y 38.522, Z 79.900}
   LaserStart_Ext()
   LIN {X -6.562, Y 38.522, Z 79.900}
   LaserEnd_Ext()
   LIN {X -6.160, Y 37.522, Z 79.900}
   LaserStart_Ext()
   LIN {X 0.655, Y 37.522, Z 79.900}
   LaserEnd_Ext()
   LIN {X 1.090, Y 36.522, Z 79.900}
   LaserStart_Ext()
   LIN {X -5.773, Y 36.522, Z 79.900}
   LaserEnd_Ext()
   LIN {X -5.399, Y 35.522, Z 79.900}
   LaserStart_Ext()
   LIN {X 1.513, Y 35.522, Z 79.900}
   LaserEnd_Ext()
   LIN {X 1.937, Y 34.522, Z 79.900}
   LaserStart_Ext()
   LIN {X -5.053, Y 34.522, Z 79.900}
   LaserEnd_Ext()
   LIN {X -4.707, Y 33.522, Z 79.900}
   LaserStart_Ext()
   LIN {X 2.359, Y 33.522, Z 79.900}
   LaserEnd_Ext()
   LIN {X 2.755, Y 32.522, Z 79.900}
   LaserStart_Ext()
   LIN {X -4.400, Y 32.522, Z 79.900}
   LaserEnd_Ext()
   LIN {X -4.124, Y 31.522, Z 79.900}
   LaserStart_Ext()
   LIN {X 3.138, Y 31.522, Z 79.900}
   LaserEnd_Ext()
   LIN {X 3.521, Y 30.522, Z 79.900}
   LaserStart_Ext()
   LIN {X -3.845, Y 30.522, Z 79.900}
   LaserEnd_Ext()
   LIN {X -3.565, Y 29.522, Z 79.900}
   LaserStart_Ext()
   LIN {X 3.860, Y 29.522, Z 79.900}
   LaserEnd_Ext()
   LIN {X 4.173, Y 28.522, Z 79.900}
   LaserStart_Ext()
   LIN {X -3.286, Y 28.522, Z 79.900}
   LaserEnd_Ext()
   LIN {X -3.007, Y 27.522, Z 79.900}
   LaserStart_Ext()
   LIN {X 4.487, Y 27.522, Z 79.900}
   LaserEnd_Ext()
   LIN {X 4.800, Y 26.522, Z 79.900}
   LaserStart_Ext()
   LIN {X -2.761, Y 26.522, Z 79.900}
   LaserEnd_Ext()
   LIN {X -2.607, Y 25.522, Z 79.900}
   LaserStart_Ext()
   LIN {X 5.113, Y 25.522, Z 79.900}
   LaserEnd_Ext()
   LIN {X 5.426, Y 24.522, Z 79.900}
   LaserStart_Ext()
   LIN {X -2.445, Y 24.522, Z 79.900}
   LaserEnd_Ext()
   LIN {X -2.269, Y 23.522, Z 79.900}
   LaserStart_Ext()
   LIN {X 5.740, Y 23.522, Z 79.900}
   LaserEnd_Ext()
   LIN {X 6.053, Y 22.522, Z 79.900}
   LaserStart_Ext()
   LIN {X -2.092, Y 22.522, Z 79.900}
   LaserEnd_Ext()
   LIN {X -1.916, Y 21.522, Z 79.900}
   LaserStart_Ext()
   LIN {X 6.381, Y 21.522, Z 79.900}
   LaserEnd_Ext()
   LIN {X 6.637, Y 20.522, Z 79.900}
   LaserStart_Ext()
   LIN {X -1.740, Y 20.522, Z 79.900}
   LaserEnd_Ext()
   LIN {X -1.563, Y 19.522, Z 79.900}
   LaserStart_Ext()
   LIN {X 6.873, Y 19.522, Z 79.900}
   LaserEnd_Ext()
   LIN {X 7.095, Y 18.522, Z 79.900}
   LaserStart_Ext()
   LIN {X -1.477, Y 18.522, Z 79.900}
   LaserEnd_Ext()
   LIN {X -1.409, Y 17.522, Z 79.900}
   LaserStart_Ext()
   LIN {X 7.311, Y 17.522, Z 79.900}
   LaserEnd_Ext()
   LIN {X 7.528, Y 16.522, Z 79.900}
   LaserStart_Ext()
   LIN {X -1.342, Y 16.522, Z 79.900}
   LaserEnd_Ext()
   LIN {X -1.274, Y 15.522, Z 79.900}
   LaserStart_Ext()
   LIN {X 7.745, Y 15.522, Z 79.900}
   LaserEnd_Ext()
   LIN {X 7.962, Y 14.522, Z 79.900}
   LaserStart_Ext()
   LIN {X -1.207, Y 14.522, Z 79.900}
   LaserEnd_Ext()
   LIN {X -1.139, Y 13.522, Z 79.900}
   LaserStart_Ext()
   LIN {X 8.179, Y 13.522, Z 79.900}
   LaserEnd_Ext()
   LIN {X 8.396, Y 12.522, Z 79.900}
   LaserStart_Ext()
   LIN {X -1.071, Y 12.522, Z 79.900}
   LaserEnd_Ext()
   LIN {X -1.029, Y 11.522, Z 79.900}
   LaserStart_Ext()
   LIN {X 8.587, Y 11.522, Z 79.900}
   LaserEnd_Ext()
   LIN {X 8.714, Y 10.522, Z 79.900}
   LaserStart_Ext()
   LIN {X -1.016, Y 10.522, Z 79.900}
   LaserEnd_Ext()
   LIN {X -1.004, Y 9.522, Z 79.900}
   LaserStart_Ext()
   LIN {X 8.841, Y 9.522, Z 79.900}
   LaserEnd_Ext()
   LIN {X 8.969, Y 8.522, Z 79.900}
   LaserStart_Ext()
   LIN {X -0.991, Y 8.522, Z 79.900}
   LaserEnd_Ext()
   LIN {X -1.056, Y 7.522, Z 79.900}
   LaserStart_Ext()
   LIN {X 9.096, Y 7.522, Z 79.900}
   LaserEnd_Ext()
   LIN {X 9.224, Y 6.522, Z 79.900}
   LaserStart_Ext()
   LIN {X -1.127, Y 6.522, Z 79.900}
   LaserEnd_Ext()
   LIN {X -1.198, Y 5.522, Z 79.900}
   LaserStart_Ext()
   LIN {X 9.351, Y 5.522, Z 79.900}
   LaserEnd_Ext()
   LIN {X 9.478, Y 4.522, Z 79.900}
   LaserStart_Ext()
   LIN {X -1.269, Y 4.522, Z 79.900}
   LaserEnd_Ext()
   LIN {X -1.331, Y 3.522, Z 79.900}
   LaserStart_Ext()
   LIN {X 9.606, Y 3.522, Z 79.900}
   LaserEnd_Ext()
   LIN {X 9.733, Y 2.522, Z 79.900}
   LaserStart_Ext()
   LIN {X -1.393, Y 2.522, Z 79.900}
   LaserEnd_Ext()
   LIN {X -1.458, Y 1.522, Z 79.900}
   LaserStart_Ext()
   LIN {X 9.868, Y 1.522, Z 79.900}
   LaserEnd_Ext()
   LIN {X 9.973, Y 0.522, Z 79.900}
   LaserStart_Ext()
   LIN {X -1.587, Y 0.522, Z 79.900}
   LaserEnd_Ext()
   LIN {X -1.766, Y -0.478, Z 79.900}
   LaserStart_Ext()
   LIN {X 10.021, Y -0.478, Z 79.900}
   LaserEnd_Ext()
   LIN {X 10.066, Y -1.478, Z 79.900}
   LaserStart_Ext()
   LIN {X -1.942, Y -1.478, Z 79.900}
   LaserEnd_Ext()
   LIN {X -2.117, Y -2.478, Z 79.900}
   LaserStart_Ext()
   LIN {X 10.111, Y -2.478, Z 79.900}
   LaserEnd_Ext()
   LIN {X 10.156, Y -3.478, Z 79.900}
   LaserStart_Ext()
   LIN {X -2.292, Y -3.478, Z 79.900}
   LaserEnd_Ext()
   LIN {X -2.468, Y -4.478, Z 79.900}
   LaserStart_Ext()
   LIN {X 10.201, Y -4.478, Z 79.900}
   LaserEnd_Ext()
   LIN {X 10.246, Y -5.478, Z 79.900}
   LaserStart_Ext()
   LIN {X -2.643, Y -5.478, Z 79.900}
   LaserEnd_Ext()
   LIN {X -2.867, Y -6.478, Z 79.900}
   LaserStart_Ext()
   LIN {X 10.243, Y -6.478, Z 79.900}
   LaserEnd_Ext()
   LIN {X 10.239, Y -7.478, Z 79.900}
   LaserStart_Ext()
   LIN {X -3.119, Y -7.478, Z 79.900}
   LaserEnd_Ext()
   LIN {X -3.372, Y -8.478, Z 79.900}
   LaserStart_Ext()
   LIN {X 10.234, Y -8.478, Z 79.900}
   LaserEnd_Ext()
   LIN {X 10.230, Y -9.478, Z 79.900}
   LaserStart_Ext()
   LIN {X -3.626, Y -9.478, Z 79.900}
   LaserEnd_Ext()
   LIN {X -3.911, Y -10.478, Z 79.900}
   LaserStart_Ext()
   LIN {X 10.212, Y -10.478, Z 79.900}
   LaserEnd_Ext()
   LIN {X 10.167, Y -11.478, Z 79.900}
   LaserStart_Ext()
   LIN {X -4.218, Y -11.478, Z 79.900}
   LaserEnd_Ext()
   LIN {X -4.523, Y -12.478, Z 79.900}
   LaserStart_Ext()
   LIN {X 10.123, Y -12.478, Z 79.900}
   LaserEnd_Ext()
   LIN {X 10.080, Y -13.478, Z 79.900}
   LaserStart_Ext()
   LIN {X 3.064, Y -13.478, Z 79.900}
   LaserEnd_Ext()
   LIN {X 0.267, Y -13.478, Z 79.900}
   LaserStart_Ext()
   LIN {X -4.862, Y -13.478, Z 79.900}
   LaserEnd_Ext()
   LIN {X -5.219, Y -14.478, Z 79.900}
   LaserStart_Ext()
   LIN {X -1.988, Y -14.478, Z 79.900}
   LaserEnd_Ext()
   LIN {X 5.068, Y -14.478, Z 79.900}
   LaserStart_Ext()
   LIN {X 10.023, Y -14.478, Z 79.900}
   LaserEnd_Ext()
   LIN {X 9.948, Y -15.478, Z 79.900}
   LaserStart_Ext()
   LIN {X 6.017, Y -15.478, Z 79.900}
   LaserEnd_Ext()
   LIN {X -2.941, Y -15.478, Z 79.900}
   LaserStart_Ext()
   LIN {X -5.578, Y -15.478, Z 79.900}
   LaserEnd_Ext()
   LIN {X -5.919, Y -16.478, Z 79.900}
   LaserStart_Ext()
   LIN {X -3.688, Y -16.478, Z 79.900}
   LaserEnd_Ext()
   LIN {X 6.720, Y -16.478, Z 79.900}
   LaserStart_Ext()
   LIN {X 9.874, Y -16.478, Z 79.900}
   LaserEnd_Ext()
   LIN {X 9.781, Y -17.478, Z 79.900}
   LaserStart_Ext()
   LIN {X 7.245, Y -17.478, Z 79.900}
   LaserEnd_Ext()
   LIN {X -3.953, Y -17.478, Z 79.900}
   LaserStart_Ext()
   LIN {X -6.119, Y -17.478, Z 79.900}
   LaserEnd_Ext()
   LIN {X -6.315, Y -18.478, Z 79.900}
   LaserStart_Ext()
   LIN {X -4.218, Y -18.478, Z 79.900}
   LaserEnd_Ext()
   LIN {X 7.376, Y -18.478, Z 79.900}
   LaserStart_Ext()
   LIN {X 9.679, Y -18.478, Z 79.900}
   LaserEnd_Ext()
   LIN {X 9.577, Y -19.478, Z 79.900}
   LaserStart_Ext()
   LIN {X 7.503, Y -19.478, Z 79.900}
   LaserEnd_Ext()
   LIN {X -4.458, Y -19.478, Z 79.900}
   LaserStart_Ext()
   LIN {X -6.399, Y -19.478, Z 79.900}
   LaserEnd_Ext()
   LIN {X -6.205, Y -20.478, Z 79.900}
   LaserStart_Ext()
   LIN {X -4.250, Y -20.478, Z 79.900}
   LaserEnd_Ext()
   LIN {X 7.326, Y -20.478, Z 79.900}
   LaserStart_Ext()
   LIN {X 9.390, Y -20.478, Z 79.900}
   LaserEnd_Ext()
   LIN {X 9.070, Y -21.478, Z 79.900}
   LaserStart_Ext()
   LIN {X 6.976, Y -21.478, Z 79.900}
   LaserEnd_Ext()
   LIN {X -4.001, Y -21.478, Z 79.900}
   LaserStart_Ext()
   LIN {X -6.016, Y -21.478, Z 79.900}
   LaserEnd_Ext()
   LIN {X -5.822, Y -22.478, Z 79.900}
   LaserStart_Ext()
   LIN {X -3.483, Y -22.478, Z 79.900}
   LaserEnd_Ext()
   LIN {X 6.614, Y -22.478, Z 79.900}
   LaserStart_Ext()
   LIN {X 8.759, Y -22.478, Z 79.900}
   LaserEnd_Ext()
   LIN {X 8.241, Y -23.478, Z 79.900}
   LaserStart_Ext()
   LIN {X 5.680, Y -23.478, Z 79.900}
   LaserEnd_Ext()
   LIN {X -2.689, Y -23.478, Z 79.900}
   LaserStart_Ext()
   LIN {X -5.196, Y -23.478, Z 79.900}
   LaserEnd_Ext()
   LIN {X -4.566, Y -24.478, Z 79.900}
   LaserStart_Ext()
   LIN {X -1.315, Y -24.478, Z 79.900}
   LaserEnd_Ext()
   LIN {X 4.448, Y -24.478, Z 79.900}
   LaserStart_Ext()
